FUNCTION_BLOCK "GCS7_E_DCOS"	// FB 43
TITLE = Scale DCOS
//  
//COPYRIGHT:    (C) 2003  BUHLER AG, CH-9240 UZWIL, SWITZERLAND
//
//PRODUCT:      GCS7
//
//TITLE:        Element Control DCOS
//
//-------------------------------------------------------------------------
//
//IDENT:        AUTHOR:             DEPT:                       DATE:
//FB43.2.2      A. Egli             BASE                        09-Apr-2008
//              Disable Alarm 18 Battery Low
//FB43.2.1      A.Egli              CT3                         01-Dec-2005
//              Parameter Upload Change DBD86-->DBD88
//FB43.2.0      A.Egli              CT3                         05-Jan-2005
//              Parameter Upload (uses DB10)
//FB43.1.3      A.Egli              CT3                         13-Apr-2004
//              Copy TotalReady only when Block 1 is read
//FB43.1.2      A.Egli              CT3                         17-Nov-2003
//              - Alarm 90: Fault not DPRemoteControl
//              - Ignor SumFault as long AlarmNr <>0
//FB43.1.1      A. Egli             CT3                         05-Aug-2003
//              Reset Par.HelpFlags.OutIngrActive
//FB43.1.0      A. Egli             CT3                         02-Apr-2003
//              1st Release in S7
//
//-------------------------------------------------------------------------
//
//PURPOSE:      MANUAL : see [DOSxxMAN]
//
//RESTRICTIONS: S7
//
//=======================================================
//Log Message: 
//------------------------------------------------------
//0     = Fault Cannceled
//1..79 = AlarmLC : Alarmnumber see manual of MEAF
//90    = Fault Remote Control
//91    = StPassive
//92    = StDosing
//93    = StEmptied
//94    = Timeout starting
//95    = WrongValue
//96    = Communication fault
//97    = 
//98    = 
//99    = Collected alarm
//
//=======================================================
//StCode:  State               
//------------------------------------------------------
//32   StFault                 
// 1   StPassive               
//41   StPassive.HWStop              StPassive + InHWStop 
//51   StPassive.DPFault             StPassive + DPFault
// 2   StStarting              
// 3   StDosing                
// 9   StEmptying              
//10   StEmptied               
//11   StRefill                
AUTHOR : EA
FAMILY : GCS7LL
NAME : DCOS
VERSION : 2.2
VAR
  StCode : INT ;	//Element state code
  InEnable : BOOL ;	//Enable to run scale
  CmdAbort : BOOL ;	//Abort ingredient
  InLocalControl : BOOL ;	//Local start and abort
  spare23 : BOOL ;
  CmdNewIngr : BOOL ;	//Start new ingredient
  In_Q_ResultIngr : BOOL ;	//Acknowledge resulting
  InEmptying : BOOL ;	//Fully emptying scale hopper
  spare27 : BOOL ;
  CmdOff : BOOL ;	//Pulse to stop scale (manual mode)
  CmdOn : BOOL ;	//Pulse to start scale(manual mode)
  spare33 : BOOL ;	//Ingredient is ready for resulting
  CmdFaultReset : BOOL ;	//Command to reset fault
  InLocal : BOOL ;	//1= Local mode (no fault by start with service switch)
  InManual : BOOL ;	//1= Manual/ 0= Automatic
  InReport : BOOL ;	//Report of all state transitions
  spare37 : BOOL ;
  InHWStop : BOOL ;	//Hardware stop
  OutEnableLocal : BOOL ;
  InSimulation : BOOL ;	//Simulation with DPSim
  Out_F_ResultIngr : BOOL ;	//Announcement resulting ingredient
  OutComFault : BOOL ;	//Communication fault
  OutEmptied : BOOL ;	//Scale hopper is empytied
  OutIngrActive : BOOL ;	//Ingredient is activele
  OutWrongValue : BOOL ;	//Wrong nominal values, rejected by MEAF
  StPassive : BOOL ;	//Element is passive, no ingredient active
  StStarting : BOOL ;	//Scale is starting
  StDosing : BOOL ;	//Scale is dosing
  StEmptying : BOOL ;	//Emptying is active
  StFault : BOOL ;	//Element has a fault
  StEmptied : BOOL ;	//Hopper is emptied
  StWaiting : BOOL ;	//Scale is waiting for next ingredient
  StSuspended : BOOL ;	//Ingredient is suspended
  InRecipeNr : INT ;	//[1..8] Is send to LC
  InWeight : DINT ;	//[DIV] Is send to LC
  OutRecipeNr : INT ;	//Is read from LC
  OutWeight : DINT ;	//[DIV] Ingredient weight, is read from scale
  OutScaleWeight : DINT ;	//[DIV] Scale weight, is read from LC
  spare : DINT ;
  OutDecimalPoint : INT ;	//Is read from LC
  OutLCStep : INT ;	//Is read from LC
  OutAlarmNr : INT ;	//Is read from LC
  OutAlarmNrLog : INT ;	//Last textnumber send to log
  Recipe : STRUCT 	//Recipe Diff Scale (Profibus only)
   InRecipeNr : INT ;	//Recipe to read or write (DIFF only)
   CmdSend : BOOL ;	//1= Send Dataset 136
   CmdRead : BOOL ;	//1= Read Dataset 136
   OutSendDone : BOOL ;	//Send is done
   OutReadDone : BOOL ;	//Read is done
   OutWrongValue : BOOL ;	//MEAF has recipe rejected
   Para : STRUCT 	//DIFF: Pre cutoff weight
    InOutBinNr : INT ;	//Bin number =REC.BIN
    InOutWeightNominal : DINT ;	//[DIV] Target weight  =REC.WTS
    InOutTolPosWeight : INT ;	//[DIV] Tolerance weight positive =REC.TOL+
    InOutTolNegWeight : INT ;	//[DIV] Tolerance weight negative =REC.TOL-
    InOutFineDosingWeight : INT ;	//[DIV] Fine dosing weight =REC.STRT
    InOutCutoffWeight : INT ;	//[DIV] Pre cutoff weight =REC.CUTW
    InOutDosingSpeedFast : INT ;	//[%] Fast dosing speed =REC.FFLO
    InOutDosingSpeedSlow : INT ;	//[%] Slow dosing speed =REC.DFLO
   END_STRUCT ;
  END_STRUCT ;
  Par : STRUCT
   ParObjectNo : INT ;	//Is used for communication with PC, e.g. for message
   ParMsgType : INT ;	//Is used for message (translation of state)
   ParHornCode : INT ;	//Is used by horn module
   ParLogOff : BOOL ;	//Report is off
   ParManual : BOOL ;	//Manual mode without interlocking
   ParPosWeighing : BOOL ;	//1=Positve weighing, 0=Negativ weighing
   ParFilter : STRUCT 	//Filter to alarm 1=Ignore alarm
    SumFault : BOOL ;	//All: de: Sammelalarm
    A05_24VToLow : BOOL ;	//All:
    A07ADRange : BOOL ;
    A08ADCalibration : BOOL ;
    A09ADFunction : BOOL ;
    A10ADSupply : BOOL ;
    A11AnalogInput : BOOL ;
    AxxCommunication : BOOL ;	//A12: Serial Interface ; A14=DPFault
    A13RemoteControl : BOOL ;
    A16Printer : BOOL ;
    A18BatteryLow : BOOL ;
    A20NoStandStill : BOOL ;
    A26Tolerance : BOOL ;
    A30ZeroTara : BOOL ;
    A42Limit : BOOL ;
    A63ProductFlow : BOOL ;
   END_STRUCT ;
   ParIOByteNr : INT ;	//PROFIBUS: Address of first input and output byte Profibus DP
   ParMonTime : INT ;	//After this time the scale must be in the requested state (New)
   Spare90 : DINT ;
   Spare94 : DINT ;
   OutMonTime : INT ;
   HelpFlags : STRUCT 	//Aux. signal to retry fault message
    OutFaultResetDone : BOOL ;
    OutTestNewAlarm : BOOL ;
    OutFlagFaultResetDone : BOOL ;
    OutAlarmTimeOut : BOOL ;
    spare : BOOL ;	//Help flag for immediate stop
    OutRelevantFault : BOOL ;
    OutNoAlarm : BOOL ;	//Alarmnumber 0 is read form LC
    OutComFaultRead : BOOL ;
    OutComFaultSend : BOOL ;
    OutIngrActive : BOOL ;
   END_STRUCT ;
   Command : STRUCT 	//Command for LC, is send to LC
    Start : BOOL ;	//de: Start
    Abort : BOOL ;	//de: Abbruch
    ControlByDP : BOOL ;	//de: Bedienung über Profibus DP
    spare03 : BOOL ;
    spare04 : BOOL ;
    spare05 : BOOL ;
    Emptying : BOOL ;	//de: Entleeren / Charge beenden
    AcceptTotalReady : BOOL ;	//de: Quittierung neue Werte Bereit
    AcceptStart : BOOL ;	//de: Quittierung 24V Start/Stop Signal
    AcceptAbort : BOOL ;	//de: Quittierung 24V Abbruch Signal
    spare20 : BYTE ;
    CommandReady : BOOL ;	//de: Steuersignale gültig
    spare41 : BOOL ;
    spare42 : BOOL ;
    spare43 : BOOL ;
    spare44 : BOOL ;
    ResetAlarm : BOOL ;	//de: Alarm löschen
    NewSendData : BOOL ;	//de: Aenderung Sendedaten
    AcceptNewRcvData : BOOL ;	//de: Quittierung Aenderung Empfangsdatensatz
   END_STRUCT ;
   Status : STRUCT 	//MEAF DIFF
    Operation : BOOL ;	//de: Betrieb
    spare01 : BOOL ;
    ReadyDosing : BOOL ;	//de: Dosierbereit
    FastDosing : BOOL ;	//de: Grobdosieren
    SlowDosing : BOOL ;	//de: Feindosieren
    Emptying : BOOL ;	//de: Entleerung aktiv
    EmptyingDone : BOOL ;	//de: Entleeren ausgefüht
    TotalReady : BOOL ;	//de: Total erreicht
    Start : BOOL ;	//de: Start/Stop 24V
    Abort : BOOL ;	//de: Abbruch 24V
    spare20 : BYTE ;
    spare30 : BOOL ;
    spare31 : BOOL ;
    spare32 : BOOL ;	//de: Stuerung Remote
    RemoteControlDP : BOOL ;	//de: Sollwertvorgabe Remote
    WrongValue : BOOL ;	//de: Falscher Sollwert
    SumFault : BOOL ;	//de: Sammelalarm
    AcceptNewSendData : BOOL ;	//de: Quittierung Aenderung Sendedaten
    NewRcvData : BOOL ;	//de: Aenderung Empfangsdaten
   END_STRUCT ;
  END_STRUCT ;
END_VAR
VAR_TEMP
  tmpLOGvalue : WORD ;	//LOG value
  tmpCommand : INT ;
  tmpReport : BOOL ;	//Global LOG all
  tmpFault : BOOL ;
  tmpLocal : BOOL ;
  tmpOn : BOOL ;
  tmpOff : BOOL ;
  tmpSeqStopDUMP : BOOL ;
  tmpWeight : DINT ;
  tmpLenDyn : DINT ;
  tmpImmediateStop : BOOL ;
  tmpFilter : ARRAY  [0 .. 100 ] OF BOOL ;
  tmpAlarmDIFF : STRUCT 	//Is read from DIFF with command d
   DepotEmpty : BOOL ;	//Surge hopper empty (not on collect alarm) --> alarm 34
   ScaleEmpty : BOOL ;	//de: Leerstand Waage (no product)
   Discharger : BOOL ;	//DIFF a2 Frequency converter or feeding drive -->alarm 25
   Tolerance : BOOL ;	//DIFF a2 Tolerance --> alarm 26
   SumFault : BOOL ;	//de: Sammelalarm ab V26A
   TaraPos : BOOL ;	//DIFF a1 n.w.  -->alarm 30
   ADConverter : BOOL ;	//DIFF a1 AD converter--> alarm 9
   Reading : BOOL ;	//DIFF a1 Measuring fault --> alarm 27
  END_STRUCT ;
  tmpAddr : WORD ;
  tmpReturn : INT ;
  DPData : STRUCT
   StatusCommand : DWORD ;
   NrSndDataSet : BYTE ;	//de: Nummer Sendedatensatz
   IdxSndDataSet : BYTE ;	//de: Index Sendedatensatz
   NrRcvDataSet : BYTE ;	//de: Nummer Empfangsdatensatz
   IdxRcvDataSet : BYTE ;	//de: Index Empfangsdatensatz
   Data : STRUCT
    Value8 : DINT ;
    Value12 : DINT ;
    Value16 : DINT ;
    Value20 : BYTE ;
    Value21 : BYTE ;
    Value22 : BYTE ;
    Value23 : BYTE ;
   END_STRUCT ;
  END_STRUCT ;
  tmpTotalReady : BOOL ;
END_VAR
BEGIN
NETWORK
TITLE =  Start Global
      L     90;
      T     #tmpLenDyn;	//--> Len dynamic data in byte
NETWORK
TITLE = Filter
      LAR1  P##tmpFilter;
      L     0;
      T     D [AR1,P#0.0];	//tmpFilter[00..31]
      T     D [AR1,P#0.0];	//tmpFilter[32..63]
      T     D [AR1,P#0.0];	//tmpFilter[64..95]
      SET;	//[1.2]
      =     #tmpFilter[0];
      A     #Par.ParFilter.A05_24VToLow;
      =     #tmpFilter[5];
      A     #Par.ParFilter.A07ADRange;
      =     #tmpFilter[7];
      A     #Par.ParFilter.A08ADCalibration;
      =     #tmpFilter[8];
      A     #Par.ParFilter.A09ADFunction;
      =     #tmpFilter[9];
      A     #Par.ParFilter.A10ADSupply;
      =     #tmpFilter[10];
      A     #Par.ParFilter.A11AnalogInput;
      =     #tmpFilter[11];
      A     #Par.ParFilter.AxxCommunication;
      =     #tmpFilter[12];
      =     #tmpFilter[14];
      A     #Par.ParFilter.A13RemoteControl;
      =     #tmpFilter[13];
      A     #Par.ParFilter.A16Printer;
      =     #tmpFilter[16];
      SET;
      =     #tmpFilter[18];	//[2.2] Battery Low
      A     #Par.ParFilter.A20NoStandStill;
      =     #tmpFilter[20];
      A     #Par.ParFilter.A26Tolerance;
      =     #tmpFilter[26];
      A     #Par.ParFilter.A30ZeroTara;
      =     #tmpFilter[30];
      A     #Par.ParFilter.A42Limit;
      =     #tmpFilter[42];
      A     #Par.ParFilter.A63ProductFlow;
      =     #tmpFilter[63];
NETWORK
TITLE = PC Control
//=== Test Object number =====================
      L     "SYS_DirectCtrlDB".PC.ObjectNo;	//PCControl.ObjectNo
      L     #Par.ParObjectNo;	//Input ObjectNo
      <>I;
      JC    Ctrl;
//=== Test OType      ========================
      L     1043;	//Input object type
      L     "SYS_DirectCtrlDB".PC.ObjectType;	//PCControl.ObjectType
      <>I;
      JC    Ctrl;
//=== Test Handshake =========================
      A     "SYS_DirectCtrlDB".PC.Hsk.FExamine;	//Handshake.FExamine
      JC    pExa;
      A     "SYS_DirectCtrlDB".PC.Hsk.FDefineCmd;	//Handshake.FDefineCmd
      JC    pCmd;
      A     "SYS_DirectCtrlDB".PC.Hsk.FDefinePara;	//Handshake.FDefinePara
      JC    pPar;
pIni: L     2;	//FcInit
      UC    "SYS_DirectCtrl";
      JU    Ctrl;
// Write parameter 
pPar: LAR1  P#DBX 58.0;
      L     P##Par;
      L     DW#16#FFFFF;
      AD;
      +AR1;
      L     DBD [AR1,P#12.0];
      T     #Par.ParMonTime;
//Write new commands from PC to Interface of group 
pCmd: A     "SYS_DirectCtrlDB".PC.Cmd1[1];	//Cmd1[1]  =CmdAbort
      S     #CmdAbort;
      A     "SYS_DirectCtrlDB".PC.Cmd1[6];	//Cmd1[2]  =CmdEmptyingOn
      S     #InEmptying;
      A     "SYS_DirectCtrlDB".PC.Cmd2[6];	//Cmd1[2]  =CmdEmptyingOff
      R     #InEmptying;
      A     "SYS_DirectCtrlDB".PC.Cmd1[4];	//Cmd1[4]  =CmdNewIngr
      S     #CmdNewIngr;
      R     #InEmptying;
      A     "SYS_DirectCtrlDB".PC.Cmd1[5];	//Cmd1[5]  =Cmd_Q_ResultIngr
      S     #In_Q_ResultIngr;
      A     "SYS_DirectCtrlDB".PC.Cmd1[8];	//Cmd1[8]  =CmdOff
      S     #CmdOff;
      A     "SYS_DirectCtrlDB".PC.Cmd1[9];	//Cmd1[9]  =CmdOn
      S     #CmdOn;
      A     "SYS_DirectCtrlDB".PC.Cmd1[11];	//Cmd1[11]=CmdFaultReset
      S     #CmdFaultReset;
      A     "SYS_DirectCtrlDB".PC.Cmd1[13];	//Cmd1[13]=CmdManualOn
      S     #InManual;
      A     "SYS_DirectCtrlDB".PC.Cmd2[13];	//Cmd2[13]=CmdManualOff
      R     #InManual;
      A     "SYS_DirectCtrlDB".PC.Cmd1[14];	//Cmd1[14]=CmdReportOn
      S     #InReport;
      A     "SYS_DirectCtrlDB".PC.Cmd2[14];	//Cmd2[14]=CmdReportOff
      R     #InReport;
//Define Value
      AN    "SYS_DirectCtrlDB".PC.Hsk.FDefineValue;	// PC.Hsk.FDefineValue
      ON    #InManual;
      JC    pIni;
      LAR1  P#DBX 58.0;
      L     DBW [AR1,P#6.0];
      T     #InRecipeNr;
      L     DBD [AR1,P#8.0];
      T     #InWeight;
      JU    pIni;
pExa: TAR2;	//Address Dynamic datas
      T     "SYS_DirectCtrlDB".GC.InDynAddr;	//-->PCControl.GC.InDynAddr
      L     #tmpLenDyn;	//Length Dynamic datas
      T     "SYS_DirectCtrlDB".GC.InDynLen;	//-->PCControl.GC.InDynLen
      L     0;
      T     "SYS_DirectCtrlDB".GC.InParaAddr;	//-->PCControl.GC.InParaAddr
      T     "SYS_DirectCtrlDB".GC.InParaLen;	//-->PCControl.GC.InParaLen
      L     1;	//Code FcExamine
      UC    "SYS_DirectCtrl";
      L     10;	//Revision
      T     "SYS_DirectCtrlDB".GC.Revision;
Ctrl: NOP   0;
NETWORK
TITLE = (Profibus) Read data
//**********************************
//(Profibus)
//**********************************
      L     #Par.ParIOByteNr;
      T     #tmpAddr;
      A     #InSimulation;
      JC    rSim;
      CALL  "SIEMENS_DPRD_DAT" (
           LADDR                    := #tmpAddr,
           RET_VAL                  := #tmpReturn,
           RECORD                   := #DPData);
      L     #tmpReturn;
      L     0;
      <>I;
      =     #Par.HelpFlags.OutComFaultRead;
      JC    rcv0;
      JU    rDP;
//read from Simulation
rSim: R     #Par.HelpFlags.OutComFaultRead;
      A     "GCS7_Gr_SimDPtoImage";
      L     P#I 0.0;
      JC    rDB1;
      OPN   "TEST_IOSimuliInput";
      L     P#DBX 0.0;
rDB1: L     #Par.ParIOByteNr;
      SLD   3;
      +D;
      LAR1;
      L     D [AR1,P#0.0];
      T     #DPData.StatusCommand;
      L     B [AR1,P#4.0];
      T     #DPData.NrSndDataSet;
      L     B [AR1,P#5.0];
      T     #DPData.IdxSndDataSet;
      L     B [AR1,P#6.0];
      T     #DPData.NrRcvDataSet;
      L     B [AR1,P#7.0];
      T     #DPData.IdxRcvDataSet;
      L     D [AR1,P#8.0];
      T     #DPData.Data.Value8;
      L     D [AR1,P#12.0];
      T     #DPData.Data.Value12;
      L     D [AR1,P#16.0];
      T     #DPData.Data.Value16;
      L     B [AR1,P#20.0];
      T     #DPData.Data.Value20;
      L     B [AR1,P#21.0];
      T     #DPData.Data.Value21;
      L     B [AR1,P#22.0];
      T     #DPData.Data.Value22;
      L     B [AR1,P#23.0];
      T     #DPData.Data.Value23;
//==Copy Status===============
rDP:  L     #DPData.NrRcvDataSet;
      L     0;
      ==I;
      JC    R001;
      A     #Par.Status.TotalReady;	//[1.3]
      =     #tmpTotalReady;	//[1.3]
      CALL  "SIEMENS_BLKMOV" (
           SRCBLK                   := #DPData.StatusCommand,
           RET_VAL                  := #tmpReturn,
           DSTBLK                   := #Par.Status);
      A     #tmpTotalReady;	//[1.3]
      =     #Par.Status.TotalReady;	//[1.3]
      AN    #Par.Status.NewRcvData;
      A     #InSimulation;
      JC    rcv0;
//===============================
//Answer Dataset 001
      L     #DPData.NrRcvDataSet;
      L     1;
      <>I;
      JC    r11;	//[2.0]
      CALL  "SIEMENS_BLKMOV" (
           SRCBLK                   := #DPData.StatusCommand,
           RET_VAL                  := #tmpReturn,
           DSTBLK                   := #Par.Status);	//[1.3]
      AN    #Par.HelpFlags.OutIngrActive;
      JC    rJ4;
      L     #DPData.Data.Value8;
      T     #OutWeight;
rJ4:  L     #DPData.Data.Value12;
      T     #OutScaleWeight;
      L     #DPData.Data.Value20;
      T     #OutDecimalPoint;
      L     #DPData.Data.Value21;
      T     #OutRecipeNr;
      L     #DPData.Data.Value22;
      T     #OutLCStep;
//Reset old alarm flags with CmdFaultReset
      A     #Par.HelpFlags.OutFlagFaultResetDone;
      A     "SYS_Pulse1000ms";
      R     #Par.HelpFlags.OutFlagFaultResetDone;
      R     #Par.HelpFlags.OutFaultResetDone;
      S     #Par.HelpFlags.OutTestNewAlarm;
      L     #DPData.Data.Value23;	//[1.2]
      L     0;	//[1.2]
      <>I;	//[1.2]
      O     #Par.ParFilter.SumFault;	//[1.2]
      =     #tmpFilter[0];	//[1.2]
      L     0;
      L     #DPData.Data.Value23;
      ==I;
      =     #Par.HelpFlags.OutNoAlarm;
//  keep old alalrm number
      A     #Par.HelpFlags.OutNoAlarm;
      A     #Par.HelpFlags.OutRelevantFault;
      AN    #Par.HelpFlags.OutTestNewAlarm;
      AN    #InLocal;
      AN    #InManual;
      JC    rA1;
      T     #OutAlarmNr;
rA1:  NOP   0;
      JU    R11;	//[2.0]   
//===============================
//[7.0]--> LC Parameter 
//Reading dataset 11
R11:  L     "SYS_DirectCtrlLCDB".PC.ObjectNo;
      L     #Par.ParObjectNo;
      <>I;
      JC    R127;
      AN    "SYS_DirectCtrlLCDB".PC.Hsk.FExamineFirst;
      AN    "SYS_DirectCtrlLCDB".PC.Hsk.FExamineNext;
      JC    R127;
// -- Start Reading with Dataset 11
      L     11;
      T     #DPData.NrRcvDataSet;
      L     253;	//First
      A     "SYS_DirectCtrlLCDB".PC.Hsk.FExamineFirst;
      JC    rLC9;
      L     254;	//Next
rLC9: T     #DPData.IdxRcvDataSet;
      JU    rcv0;
//---Answer  dataset 11 ---
//---Answer  dataset 12 ---
r11:  L     #DPData.NrRcvDataSet;
      L     11;
      <>I;
      JC    rLCB;
// Answer Dataset 11
      L     '  ';
      T     "SYS_DirectCtrlLCDB".PC.Value[1];
      L     #DPData.Data.Value8;
      T     DB10.DBD 60;
      L     #DPData.Data.Value12;
      T     DB10.DBD 64;
      L     #DPData.Data.Value16;
      T     DB10.DBD 68;
      L     #DPData.Data.Value20;
      SLD   24;
      L     #DPData.Data.Value21;
      SLD   16;
      OD;
      L     #DPData.Data.Value22;
      SLD   8;
      OD;
      L     #DPData.Data.Value23;
      OD;
      T     DB10.DBD 72;
      L     #DPData.IdxRcvDataSet;
      L     255;
      ==I;
      JC    rLCE;
      S     "SYS_DirectCtrlLCDB".GC.Set11Done;
      L     12;
      T     #DPData.NrRcvDataSet;
      L     0;
      T     #DPData.IdxRcvDataSet;
      JU    rcv0;	//--> Read dataset 12
// Answer Dataset 12
rLCB: L     #DPData.NrRcvDataSet;
      L     12;
      <>I;
      JC    r127;
      L     #DPData.Data.Value8;
      T     DB10.DBD 76;
      L     #DPData.Data.Value12;
      T     DB10.DBD 80;
      L     #DPData.Data.Value16;
      T     DB10.DBD 84;
      L     #DPData.Data.Value20;
      SLD   24;
      L     #DPData.Data.Value21;
      SLD   16;
      OD;
      L     #DPData.Data.Value22;
      SLD   8;
      OD;
      L     #DPData.Data.Value23;
      OD;
      T     DB10.DBD 88;
      AN    "SYS_DirectCtrlLCDB".GC.Set11Done;
      JC    R127;
rLCE: L     12;
      CALL  "SYS_DirectCtrl";
      JU    R127;
//<--[2.0]
//===============================
//Answer  dataset 127
r127: L     #DPData.NrRcvDataSet;
      L     127;
      <>I;
      JC    r128;
      JU    R128;
//===============================
//Answer  dataset 128
r128: L     #DPData.NrRcvDataSet;
      L     128;
      <>I;
      JC    r136;
      JU    R001;
//===============================
//Answer  dataset 136
r136: L     #DPData.NrRcvDataSet;
      L     136;
      <>I;
      JC    R001;	// =no valide answer read dataset 001
      L     #Recipe.InRecipeNr;
      L     #DPData.IdxRcvDataSet;
      ==I;
      JCN   R001;
      S     #Recipe.OutReadDone;
      R     #Recipe.CmdRead;
      CALL  "SIEMENS_BLKMOV" (
           SRCBLK                   := #DPData.Data,
           RET_VAL                  := #tmpReturn,
           DSTBLK                   := #Recipe.Para);
      L     #DPData.Data.Value22;
      T     #Recipe.Para.InOutDosingSpeedFast;
      L     #DPData.Data.Value23;
      T     #Recipe.Para.InOutDosingSpeedSlow;
      JU    R001;
//===============================
//Read Dataset 001
R001: L     1;
      T     #DPData.NrRcvDataSet;
      L     0;
      T     #DPData.IdxRcvDataSet;
      A     #Par.HelpFlags.OutFaultResetDone;
      AN    "SYS_Pulse1000ms";
      S     #Par.HelpFlags.OutFlagFaultResetDone;
      JU    rcv0;
//===============================
//Read Dataset 127
R127: L     127;
      T     #DPData.NrRcvDataSet;
      L     0;
      T     #DPData.IdxRcvDataSet;
      JU    rcv0;
//===============================
//Read Dataset 128
R128: JU    R136;
      JU    rcv0;
//===============================
//Read Dataset 136
R136: AN    #Recipe.CmdRead;
      JC    R001;
      L     136;
      T     #DPData.NrRcvDataSet;
      L     #Recipe.InRecipeNr;
      T     #DPData.IdxRcvDataSet;
rcv0: NOP   0;
      A     #Par.HelpFlags.OutComFaultRead;
      O     #Par.HelpFlags.OutComFaultSend;
      =     #OutComFault;
      NOP   0;
NETWORK
TITLE = Local Control
// ---Abort
      A     #Par.Status.Abort;
      A     #InLocalControl;
      S     #CmdAbort;
// -- Start Ingredient
      A     #Par.Status.Start;
      AN    #Par.Command.AcceptStart;
      A     #Par.Status.ReadyDosing;
      A     #InLocalControl;
      AN    #OutIngrActive;
      S     #CmdNewIngr;
      S     #OutEnableLocal;
// -- Start Local
      A     #Par.Status.Start;
      AN    #Par.Command.AcceptStart;
      AN    #OutEnableLocal;
      S     #OutEnableLocal;
      JC    aiL1;
// -- Stop Local
      A     #Par.Status.Start;
      AN    #Par.Command.AcceptStart;
      A     #OutEnableLocal;
      AN    #CmdNewIngr;
      O     #Par.Status.Abort;
      ON    #InLocalControl;
      O;
      AN    #OutIngrActive;
      AN    #CmdNewIngr;
      R     #OutEnableLocal;
aiL1: NOP   0;
NETWORK
TITLE =  All State Init
      NOP   0;
//===Global Group Orders===
      A     "GCS7_Gr_OutManualOn";	//Gr.OutManualOn
      S     #InManual;
      A     "GCS7_Gr_OutManualOff";	//Gr.OutManualOff
      R     #InManual;
      A     #InManual;
      S     "GCS7_Gr_InManual";	//Gr.InManualMode
      A     "GCS7_Gr_OutFaultReset";	//Gr.OutOutFaultReset
      O     #CmdAbort;
      S     #CmdFaultReset;
//---Report is on---
      A     "GCS7_Gr_OutReportAll";	//Gr.OutReportAll
      O     #InReport;
      =     #tmpReport;
//---Local---
      A     #InLocal;
      AN    #InManual;
      =     #tmpLocal;
//---Enable---
// tmpOff
      AN    #InEnable;
      AN    #Par.ParManual;	// 2C: U -> UN
      A     #InManual;
      O;
      AN    #InEnable;
      AN    #InManual;
      O     #CmdOff;
      O     #tmpLocal;
      O(;
      A     #InLocalControl;
      AN    #OutEnableLocal;
      );
      O     #InHWStop;
      =     #tmpOff;
      R     #OutEnableLocal;
//---On---
      AN    #InManual;
      O     #CmdOn;
      AN    #tmpOff;
      =     #tmpOn;
//--- Init in local mode  
      AN    #tmpLocal;
      JC    alJL;
      R     #OutComFault;
alJL: NOP   0;
//--- Fault   
      LAR1  P##tmpFilter;
      L     #OutAlarmNr;
      +AR1;	//Pointer to #tmpFilter[OutAlarmNumber]
      L     #OutAlarmNr;
      L     0;
      <>I;
      AN    L [AR1,P#0.0];	//#tmpFilter[OutAlarmNumber]
      O;
      A     #Par.Status.SumFault;
      AN    #tmpFilter[0];
      =     #Par.HelpFlags.OutRelevantFault;
      A     #Par.HelpFlags.OutRelevantFault;
      O     #OutComFault;
      O     #OutWrongValue;
      ON    #Par.Status.RemoteControlDP;	//[1.2]
      AN    #tmpLocal;
      =     #tmpFault;
//-- Ingredient done
      A     #Out_F_ResultIngr;
      A     #In_Q_ResultIngr;
      R     #OutIngrActive;
      A     #CmdAbort;
      O     #Par.Status.TotalReady;
      A     #OutIngrActive;
      AN    #In_Q_ResultIngr;
      =     #Out_F_ResultIngr;
//-----------------------
      A     #CmdNewIngr;
      R     #Out_F_ResultIngr;
      R     #In_Q_ResultIngr;
      R     #OutIngrActive;
      R     #Par.HelpFlags.OutIngrActive;	//[1.1]
//--Reset Actual weight during start
      A     #Par.Status.FastDosing;
      O     #Par.Status.SlowDosing;
      O     #Out_F_ResultIngr;
      S     #Par.HelpFlags.OutIngrActive;
      AN    #CmdNewIngr;
      JC    alJ2;
      L     0;
      T     #OutWeight;
//--- Recipe
alJ2: A     #Recipe.CmdRead;
      R     #Recipe.OutReadDone;
      A     #Recipe.CmdSend;
      R     #Recipe.OutSendDone;
//---Abort if Local
      A     #tmpLocal;
      A     #OutIngrActive;
      S     #CmdAbort;
      R     #CmdNewIngr;
      A     #Par.Status.ReadyDosing;
      A     #tmpLocal;
      R     #OutIngrActive;
NETWORK
TITLE = Monitoring [6.0]
//Monitoring Time [6.0]
      A     #StPassive;
      O     #CmdFaultReset;
      R     #Par.HelpFlags.OutAlarmTimeOut;	//[6.0]
      AN    #StStarting;	//[6.0]
      JC    mtJ0;	//[6.0]
      ON    "GCS7_Gr_OutTick200ms";	//[6.0]
      JC    mtJ1;	//[6.0]
      L     #Par.OutMonTime;	//[6.0]
      +     -2;	//[6.0]
      T     #Par.OutMonTime;	//[6.0]
      L     0;	//[6.0]
      >=I;	//[6.0]
      JC    mtJ1;	//[6.0]
      S     #Par.HelpFlags.OutAlarmTimeOut;	//[6.0]
      JU    mtJ1;	//[6.0]
mtJ0: L     #Par.ParMonTime;	//[6.0]
      T     #Par.OutMonTime;	//[6.0]
mtJ1: NOP   0;
NETWORK
TITLE = States
//===State machine===
      A     #StPassive;
      JC    S0;
      A     #StStarting;
      JC    S1;
      A     #StDosing;
      JC    S2;
      A     #StEmptying;
      JC    S3;
      A     #StFault;
      JC    S4;
      A     #StEmptied;
      JC    S5;
      A     #StWaiting;
      JC    S6;
      A     #StSuspended;
      JC    S7;
      S     #StPassive;	//Init
NETWORK
TITLE = StPassive
//Transition to StPassive
//Transition
xxS0: S     #StPassive;
      JU    LOGX;
//----------------------------------------------
//Logic
//Condition for StFault
S0:   A     #tmpFault;
      R     #StPassive;
      JC    xxS4;
//StEmptying
      AN    #tmpOff;
      A     #InEmptying;
      R     #StPassive;
      JC    xxS3;
//Condition for StStarting
      AN    #Par.Command.Abort;
      A     #CmdNewIngr;
      AN    #tmpOff;
      A     #Par.Status.ReadyDosing;
      AN    #Par.Status.TotalReady;
      AN    #Par.Command.AcceptTotalReady;
      R     #StPassive;
      JC    xxS1;
      JU    OUT;
NETWORK
TITLE =  STARTING
// Any Transition
//Transition
xxS1: S     #StStarting;
      S     #OutIngrActive;
      R     #CmdNewIngr;
      R     #OutEmptied;
      JU    OUT;
//----------------------------------------------
//Logic
S1:   NOP   0;
//Condition for StFault
      A     #tmpFault;
      O     #Par.HelpFlags.OutAlarmTimeOut;	//Monitoring Time [6.0]
      R     #StStarting;
      JC    xxS4;
//-- Transition to StDosing --         
      A     #Par.Status.Operation;
      AN    #OutComFault;	//[1.2]
      R     #StStarting;
      JC    xxS2;
//Condition for StSuspended
      A     #tmpOff;
      R     #StStarting;
      JC    xxS7;
//Condition for StWaiting
      AN    #OutIngrActive;
      R     #StStarting;
      JC    xxS6;
      JU    OUT;
NETWORK
TITLE =  DOSING
//Transition
//----------------------------------------------
xxS2: SET;
      S     #StDosing;
      JU    LOGX;
//----------------------------------------------
//Condition for StWaiting
S2:   AN    #OutIngrActive;
      R     #StDosing;
      JC    xxS6;
//Condition for StSuspended
      AN    #Par.Command.Start;
      O     #OutComFault;	//[1.2]
      R     #StDosing;
      JC    xxS7;
//Monitoring Time [6.0]
      A     #Par.HelpFlags.OutAlarmTimeOut;	//[6.0]
      R     #StDosing;	//[6.0]
      JC    xxS4;	//[6.0]
//Condition for Fault
      A     #tmpFault;
      R     #StDosing;
      JC    xxS4;
      JU    OUT;
NETWORK
TITLE =  FAULT
      NOP   0;
//Fault cancelled
S4:   A     #Par.HelpFlags.OutTestNewAlarm;
      AN    #tmpFault;
      O     #tmpLocal;
      JC    S4xx;
      A     #Par.HelpFlags.OutTestNewAlarm;	//[2.3] Relog fault
      A     #tmpFault;	//[2.3]
      JC    xxS4;	//[2.3]
      JU    OUT;
//Transition to StSuspended
S4xx: A     #OutIngrActive;
      R     #StFault;
      S     #StSuspended;
      JC    LOG2;	//-->//Message ('fault cancelled')
//Transition to StWaiting 
      R     #StFault;
      S     #StWaiting;
      JU    LOG2;	//-->//Message ('fault cancelled')
NETWORK
TITLE =  StEmptying
//Transition
//----------------------------------------------
xxS3: S     #StEmptying;
      JU    OUT;
//----------------------------------------------
// Condition for fault
S3:   A     #tmpFault;
      R     #StEmptying;
      JC    xxS4;
//Condition for emptied
      L     #OutScaleWeight;
      L     0;
      ==I;
      O     #Par.Status.EmptyingDone;
//     O     #Par.Status.TotalReady
      ON    #Par.ParPosWeighing;
      R     #StEmptying;
      JC    xxS5;	//-->StEmptied
//[4.0->] Back to Stopped if not emptying
      AN    #InEmptying;
      R     #StEmptying;	//avoid setting of OutEmptied
      R     #InEmptying;
      JC    xxS0;	//[<-4.0]
      JU    OUT;
NETWORK
TITLE =  StEmptied
//Condition for fault
//Transition
//----------------------------------------------
xxS5: S     #StEmptied;
      S     #OutEmptied;
      JU    LOGX;
//----------------------------------------------
S5:   A     #tmpFault;
      R     #StEmptied;
      JC    xxS4;
//Condition for Starting/Waiting
      A     #CmdNewIngr;
      R     #StEmptied;
      JC    xxS6;
//Condition for Stopped
      AN    #InEmptying;
      O     #tmpOff;
      R     #StEmptied;
      JC    xxS0;
      JU    OUT;
NETWORK
TITLE = StWaiting
//Transition
xxS6: S     #StWaiting;
      JU    OUT;
//----------------------------------------------
//Condition for fault
S6:   A     #tmpFault;
      R     #StWaiting;
      JC    xxS4;
//Condidition for StPassive
      A     #tmpLocal;
      ON    #Par.ParPosWeighing;
      R     #StWaiting;
      JC    xxS0;
//Condition for Starting
      A     #CmdNewIngr;
      AN    #Par.Command.Abort;
      AN    #Par.Status.TotalReady;
      AN    #Par.Command.AcceptTotalReady;
      R     #StWaiting;
      JC    xxS1;
//Condition for StEmptying
      A     #InEmptying;
      R     #StWaiting;
      JC    xxS3;
      JU    OUT;
NETWORK
TITLE = StSuspended
//Transition
xxS7: S     #StSuspended;
      JU    OUT;
//----------------------------------------------
//Condition for fault
S7:   A     #tmpFault;
      R     #StSuspended;
      JC    xxS4;
//Condition for Starting
      A     #Par.Command.Start;
      AN    #OutComFault;	//[1.2]
      A     #OutIngrActive;
      AN    #CmdAbort;
      R     #StSuspended;
      JC    xxS1;
//Condition for StWaiting
      AN    #OutIngrActive;
      R     #StSuspended;
      JC    xxS6;
      JU    OUT;
NETWORK
TITLE = LOG
////[5.0] Alarmnummer
xxS4: S     "GCS7_Gr_InFaultFlag";	//Gr.InFaultFlag
      S     #StFault;
//Horn On
      CALL  "SYS_Horn_Code" (
           FcCode                   := 1,
           ParObjectType            := 1040,
           ParObjectNo              := #Par.ParObjectNo,
           ParHornCode              := #Par.ParHornCode);
//Alarm Communication
      L     B#(1, 96);
      A     #OutComFault;
      JC    LOG;
//Tiemout
      A     #Par.HelpFlags.OutAlarmTimeOut;
      L     B#(1, 97);	// Message ('fault timeout')
      JC    LOG;
//Alarm-Nr 1..80
      L     0;
      L     #OutAlarmNr;
      ==I;
      JC    LOG1;
      L     B#(1, 0);
      OW;
      JU    LOG;	//Alarms 1..80
//Fault Remote Control
LOG1: L     B#(1, 90);	// Message ('fault DP Mode')   //[1.2]
      AN    #Par.Status.RemoteControlDP;	//[1.2]
      JC    LOG;	//[1.2]
//Wrong Value
      A     #OutWrongValue;
      L     B#(1, 95);	// Message ('fault wrong value')
      JC    LOG;
//Collected Alarm
      L     B#(1, 99);	// Message ('fault collected alarm')
      JU    LOG;
//Fault Cancelled
LOG2: L     B#(4, 0);	// Message ('fault collected alarm')
      JU    LOG;
//===============================================
//State Transition
LOGX: AN    #tmpReport;
      JC    OUT;
      A     #StPassive;
      L     B#(4, 91);	//Message ('Passive')
      JC    LOG;
      A     #StDosing;
      L     B#(4, 92);	//Message ('Dosing')
      JC    LOG;
      A     #StEmptied;
      L     B#(4, 93);	//Message ('Waiting')
      JC    LOG;
      A     #StEmptied;
      L     B#(4, 94);	//Message ('Emptied')
      JC    LOG;
      JU    OUT;
LOG:  A     #Par.ParLogOff;	//---Set LOG Message
      JC    OUT;
      T     #tmpLOGvalue;
      L     W#16#FF;
      AW;
      T     #OutAlarmNrLog;
      CALL  "GCS7_LogConvert" (
           ObjectNo                 := #Par.ParObjectNo,
           MsgType                  := #Par.ParMsgType,
           ClassMsgTxt              := #tmpLOGvalue,
           OType                    := 1043);	//LOG Message Converter / Entry / Contains Class and TextNo
OUT:  NOP   0;
NETWORK
TITLE = Prepare Command for MEAF
      NOP   0;
//==============================
//Abort
      A     #CmdNewIngr;
      O     #CmdAbort;
      O     #tmpLocal;
      AN    #Par.Status.TotalReady;
      A     #Par.Status.Operation;
      AN    #Par.Status.ReadyDosing;
      =     #Par.Command.Abort;
      AN    #Par.Status.Operation;
      O     #Par.Status.ReadyDosing;
      AN    #OutIngrActive;
      R     #CmdAbort;
//==============================
//  Start/Stop
      A     #StSuspended;
      A     #tmpOn;
      O     #StStarting;
      O     #StDosing;
      AN    #tmpOff;
      AN    #Par.Status.TotalReady;
      AN    #Par.Command.Abort;
      =     #Par.Command.Start;
//==============================
      SET;
      =     #Par.Command.ControlByDP;
//==============================
      L     #OutLCStep;
      L     1;
      >I;
      O     #StEmptying;
      A     #InEmptying;
      =     #Par.Command.Emptying;
//==============================
      A     #CmdAbort;
      O     #CmdFaultReset;
      AN    #Par.Status.AcceptNewSendData;
      S     #Par.Command.ResetAlarm;
      R     #CmdFaultReset;
      A     #Par.Status.AcceptNewSendData;
      A     #Par.Command.ResetAlarm;
      R     #Par.Command.ResetAlarm;
      S     #Par.HelpFlags.OutFaultResetDone;
//==============================
      A     #In_Q_ResultIngr;
      ON    #OutIngrActive;
      A     #Par.Status.TotalReady;
      =     #Par.Command.AcceptTotalReady;
//==============================
      A     #Par.Status.Start;
      =     #Par.Command.AcceptStart;
//==============================
      A     #Par.Status.Abort;
      =     #Par.Command.AcceptAbort;
//==============================
      L     #OutLCStep;
      L     8;
      <>I;
      O     "SYS_Pulse1000ms";
      ON    #Par.Status.EmptyingDone;
      =     #Par.Command.CommandReady;
//==============================
      A     #Par.Status.NewRcvData;
      =     #Par.Command.AcceptNewRcvData;
//==============================
      AN    #Par.Status.AcceptNewSendData;
      =     #Par.Command.NewSendData;
NETWORK
TITLE = Global End
      SET;	//---Clear commands
      R     #CmdOn;
      R     #Par.HelpFlags.OutTestNewAlarm;
      R     #CmdOff;
      NOP   0;
//--Output for group 
      A     #StFault;
      S     "GCS7_Gr_InFault";	// Gr.InFault
NETWORK
TITLE = (Profibus) Send Data
//Test Send Dataset 000 done
      L     #DPData.NrSndDataSet;
      L     0;
      <>I;
      JC    s128;
      JU    S128;	//-->send 128
//------------------------------------------------
//Test Send Dataset 128 done
s128: L     #DPData.NrSndDataSet;
      L     128;
      <>I;
      JC    s136;
      A     #Par.Status.WrongValue;
      =     #OutWrongValue;
      JU    S136;	//-->Send 136
//------------------------------------------------
//Test Send Dataset 129,136 done
s136: L     #DPData.NrSndDataSet;
      L     136;
      <>I;
      JC    S000;
      L     #DPData.IdxSndDataSet;
      L     #Recipe.InRecipeNr;
      ==I;
      JCN   S128;	//-->Send 128
      AN    #Par.Status.WrongValue;
      R     #Recipe.CmdSend;
      =     #Recipe.OutSendDone;
      A     #Par.Status.WrongValue;
      =     #Recipe.OutWrongValue;
      JU    S128;	//-->Send 128
//==================================================
//Send Dataset 128
S128: L     128;
      T     #DPData.NrSndDataSet;
      L     0;
      T     #DPData.IdxSndDataSet;
      L     #InWeight;
      T     #DPData.Data.Value8;
      L     0;
      T     #DPData.Data.Value12;
      T     #DPData.Data.Value16;
      T     #DPData.Data.Value20;
      T     #DPData.Data.Value21;
      T     #DPData.Data.Value22;
      T     #DPData.Data.Value23;
      L     #InRecipeNr;
      T     #DPData.Data.Value21;
      JU    Snd;
//======================================================
//Send Dataset 136
S136: A     #Recipe.CmdSend;
      JCN   S000;
      L     136;
      T     #DPData.NrSndDataSet;
      L     #Recipe.InRecipeNr;
      T     #DPData.IdxSndDataSet;
      CALL  "SIEMENS_BLKMOV" (
           SRCBLK                   := #Recipe.Para,
           RET_VAL                  := #tmpReturn,
           DSTBLK                   := #DPData.Data);
      L     #Recipe.Para.InOutDosingSpeedFast;
      T     #DPData.Data.Value22;
      L     #Recipe.Para.InOutDosingSpeedSlow;
      T     #DPData.Data.Value23;
      JU    Snd;
//======================================================
//Send Dataset 0
S000: L     0;
      T     #DPData.NrSndDataSet;
      L     0;
      T     #DPData.IdxSndDataSet;
//======================================================
//Senden DP
Snd:  CALL  "SIEMENS_BLKMOV" (
           SRCBLK                   := #Par.Command,
           RET_VAL                  := #tmpReturn,
           DSTBLK                   := #DPData.StatusCommand);
      A     #InSimulation;
      JC    sSim;
      CALL  "SIEMENS_DPWR_DAT" (
           LADDR                    := #tmpAddr,
           RECORD                   := #DPData,
           RET_VAL                  := #tmpReturn);
      L     #tmpReturn;
      L     0;
      <>I;
      =     #Par.HelpFlags.OutComFaultSend;
      JU    sEnd;
//write to Simulation
sSim: R     #Par.HelpFlags.OutComFaultSend;
      A     "GCS7_Gr_SimDPtoImage";
      L     P#Q 0.0;
      JC    rDB2;
      OPN   "TEST_IOSimuliOutput";
      L     P#DBX 0.0;
rDB2: L     #Par.ParIOByteNr;
      SLD   3;
      +D;
      LAR1;
      L     #DPData.StatusCommand;
      T     D [AR1,P#0.0];
      L     #DPData.NrSndDataSet;
      T     B [AR1,P#4.0];
      L     #DPData.IdxSndDataSet;
      T     B [AR1,P#5.0];
      L     #DPData.NrRcvDataSet;
      T     B [AR1,P#6.0];
      L     #DPData.IdxRcvDataSet;
      T     B [AR1,P#7.0];
      L     #DPData.Data.Value8;
      T     D [AR1,P#8.0];
      L     #DPData.Data.Value12;
      T     D [AR1,P#12.0];
      L     #DPData.Data.Value16;
      T     D [AR1,P#16.0];
      L     #DPData.Data.Value20;
      T     B [AR1,P#20.0];
      L     #DPData.Data.Value21;
      T     B [AR1,P#21.0];
      L     #DPData.Data.Value22;
      T     B [AR1,P#22.0];
      L     #DPData.Data.Value23;
      T     B [AR1,P#23.0];
sEnd: NOP   0;
      NOP   0;
NETWORK
TITLE = State Code
//--Passive ---
      L     41;	//Code: Passive.HWStop
      A     #InHWStop;
      A     #StPassive;
      JC    STC;
      L     1;	//Code: Passive
      A     #StPassive;
      JC    STC;
      L     2;	//Code: starting
      A     #StStarting;
      JC    STC;
      L     3;	//Code: dosing
      A     #StDosing;
      JC    STC;
      L     14;	//Code: Suspended.Resulting
      A     #StSuspended;
      A     #Out_F_ResultIngr;
      JC    STC;
      L     44;	//Code: Suspended.HWStop
      A     #InHWStop;
      A     #StSuspended;
      JC    STC;
      L     4;	//Code: Suspended
      A     #StSuspended;
      JC    STC;
      L     5;	//Code: waiting
      A     #StWaiting;
      JC    STC;
      L     9;	//Code: emptying
      A     #StEmptying;
      JC    STC;
      L     10;	//Code: emptied
      A     #StEmptied;
      JC    STC;
      L     32;	//Code: fault
STC:  L     #StCode;	//Old state code
      TAK;
      T     #StCode;	//Save state code
      <>I;
      L     3;	//Load code for CBit methode
      CC    "SYS_CBitCtrl";
END_FUNCTION_BLOCK

FUNCTION_BLOCK "GCS7_M_Scourer"	// FB 44
TITLE = Scourer
//  
//COPYRIGHT:    (C) 1997  BUHLER AG, CH-9240 UZWIL, SWITZERLAND
//
//PRODUCT:      GCS7
//
//TITLE:        FB 44 Machine Control:Scourer 
//
//-------------------------------------------------------------------------
//
//IDENT:        AUTHOR:             DEPT:                       DATE:
//
//FB44.5.6      A. Egli             CT3                         30-Aug-2009
//              Manual mode if Bypassed
//FB44.5.5      K. Tischer          CT3                         13-Feb-2004
//              - StBypassed-->StStopping
//FB44.5.4      A. Egli             CT3                         24-Nov-2003
//              - Condition for Started
//FB44.5.3      A. Egli             CT3                         11-Nov-2003
//              - StStopping-->StBypassed
//              - StStarted -->StStopping
//FB44.5.2      A. Egli             CT3                         12-Sep-2003
//              No command Scourer.CmdNext as long InSeqStop
//FB44.5.1      A. Egli             CT3                         22-Jul-2003
//              Scourer.InLocal 
//FB44.5.0      A. Egli             CT3                         17-Jun-2002
//              New Release with one block 
//FB44.4.3      Ph. Engler          MU664                       03-Apr-2002
//              - Transition from stBypassed to stStarted
//                only if Flap.StHn
//              - Scourer.InLocal reset only if not Flap.StHn
//FB44.4.2      A. Egli             CT3                         24-Mai-2002
//              Set Scourer to local, if machine is bypassed
//FB44.4.1      Ph. Engler          MU664                       13-Mar-2002
//              - Screw: CmdFaultReset corrected
//              - Machine: stFault corrected
//              - Screw: InSeqStop if bypassed integrated
//FB44.4.0      A. Egli             CT3                         24-Mai-2000
//              Screw and Scraper 
//FB44.3.1      S.Kalberer          CT3                         10-Dec-1999
//              Scourer motor seqstops on Aspiration fan fault
//FB44.3.0      A. Egli             CT3                         11-Oct-1999
//              Local data reduced 
//FB44.2B       K. Tischer          MU664                       06-Mrz-1999
//              CC FC2 not UC FC2
//FB44.2A       A. Egli             CT3                         04-Mai-1998
//              StFault = StCode 32
//FB44.1A       A.Egli              AEE61                       12-Nov-1997
//              1st Release in S7
//
//-------------------------------------------------------------------------
//
//PURPOSE:      MANUAL : see [LL.MHXENMAN]
//
//RESTRICTIONS: S7
//              ACCU2: Pointer to dynamic datas of the machine
//              ACCU1: Pointer to parameter datas of the machine
//
//-------------------------------------------------------------------------
//
//
AUTHOR : EA
FAMILY : GCS7LL
NAME : Scourer
VERSION : 5.6
VAR
  Ma : UDT 20440;
  AspLow : FB 12;	//Element
  AspHigh : FB 12;	//Element
  Scourer : FB 12;	//Element
  ManFlap : FB 13;	//Element
  HL : FB 14;	//Element
  Screw : FB 12;	//Element
  Scraper : FB 11;	//Element
END_VAR
VAR_TEMP
  tmpFaultStop : BOOL ;
  tmpFaultSum : BOOL ;
  tmpStopped : BOOL ;
  tmpOffsetInstanzDB : DWORD ;
  tmpAddrParMa : DWORD ;	//Byte Nr of first Parameter in Instanz DB
  tmpAddrParaElement : DWORD ;
  tmpNext : BOOL ;
  tmpLocal : BOOL ;
  tmpEnable : BOOL ;
  tmpEnableOpen : BOOL ;
  tmpEmpty : BOOL ;
  tmpLenDyn : INT ;
  tmpStarted : BOOL ;	//all elemenet started , without Scourer
  StoreGrOutManualOff : BOOL ;
END_VAR
BEGIN
NETWORK
TITLE =
      L     10;
      T     #tmpLenDyn;
NETWORK
TITLE = PC Control
//=== Test Object number =====================
      L     "SYS_DirectCtrlDB".PC.ObjectNo;	//PCControl.ObjectNo
      L     #Ma.Par.ParObjectNo;	//Input ObjectNo
      <>I;
      JC    aEnd;
//=== Test OType      ========================
      L     2044;	//Input object type
      L     "SYS_DirectCtrlDB".PC.ObjectType;	//PCControl.ObjectType
      <>I;
      JC    aEnd;
//=== Test Handshake =========================
      A     "SYS_DirectCtrlDB".PC.Hsk.FExamine;	// Handshake.FExamine
      JC    aExa;
      A     "SYS_DirectCtrlDB".PC.Hsk.FDefineCmd;	// Handshake.FDefineCmd
      O     "SYS_DirectCtrlDB".PC.Hsk.FDefinePara;	// Handshake.FDefinePara
      JC    aCmd;
aIni: L     2;	// FcInit
      UC    "SYS_DirectCtrl";
      JU    aEnd;
// Write new commands from PC to Interface of group 
aCmd: A     "SYS_DirectCtrlDB".PC.Cmd1[8];	//Cmd1[8]=CmdOff
      S     #Ma.CmdOff;
      A     "SYS_DirectCtrlDB".PC.Cmd1[9];	//Cmd1[9]=CmdOn
      S     #Ma.CmdOn;
      A     "SYS_DirectCtrlDB".PC.Cmd1[10];	//Cmd1[10]=CmdNext
      S     #Ma.CmdNext;
      A     "SYS_DirectCtrlDB".PC.Cmd1[11];	//Cmd1[11]=CmdFaultReset
      S     #Ma.CmdFaultReset;
      A     "SYS_DirectCtrlDB".PC.Cmd1[13];	//Cmd1[13]=CmdManualOn
      S     #Ma.InManual;
      A     "SYS_DirectCtrlDB".PC.Cmd2[13];	//Cmd1[13]=CmdManualOff
      R     #Ma.InManual;
      AN    "SYS_DirectCtrlDB".PC.Hsk.FDefinePara;	// Handshake.FDefinePara
      JC    aIni;
      JU    aIni;
aExa: TAR2;	// Address Dynamic data
      T     "SYS_DirectCtrlDB".GC.InDynAddr;	// -->PCControl.GC.InDynAddr
      L     #tmpLenDyn;	// Length Dynamic data
      T     "SYS_DirectCtrlDB".GC.InDynLen;	// -->PCControl.GC.InDynLen
      L     0;
      T     "SYS_DirectCtrlDB".GC.InParaAddr;	// -->PCControl.GC.InParaAddr
      T     "SYS_DirectCtrlDB".GC.InParaLen;	// -->PCControl.GC.InParaLen
      L     1;	// Code FcExamine
      UC    "SYS_DirectCtrl";
      L     10;	//Revision
      T     "SYS_DirectCtrlDB".GC.Revision;
aEnd: NOP   0;
NETWORK
TITLE = Interlocking
//===Global Group Orders===
      A     "GCS7_Gr_OutManualOn";	//Gr.OutManualOn
      S     #Ma.InManual;
      A     "GCS7_Gr_OutManualOff";	//Gr.OutManualOff
      R     #Ma.InManual;
      A     #Ma.InManual;
      S     "GCS7_Gr_InManual";	//Gr.InManual
      A     #Ma.CmdNext;
      AN    #Ma.InManual;
      O     #Ma.CmdOn;
      =     #tmpNext;
      A     #Ma.InLocal;
      AN    #Ma.InManual;
      =     #tmpLocal;
      AN    #tmpLocal;
      A     #Ma.InEnable;
      AN    #Ma.CmdOff;
      =     #tmpEnable;
//--- Fault----
      A     #AspLow.StFault;
      O     #AspHigh.StFault;
      O;
      A     #Scourer.StFault;	// [5.6]
      AN    #ManFlap.StHN;	// [5.6]
      O     #HL.StFault;
      O     #ManFlap.StFault;
      O     #Screw.StFault;	// [4.1]
      O     #Scraper.StFault;	// [4.1]
      =     #tmpFaultSum;
//--- Next
      AN    #Ma.Par.ParWithScrew;
      JC    InX1;
      A     #tmpNext;
      S     #Screw.CmdNext;
InX1: AN    #Ma.Par.ParWithScraper;
      JC    InX2;
      A     #tmpNext;
      S     #Scraper.CmdNext;
InX2: A(;
      O     #Screw.StStartedFwd;
      ON    #Ma.Par.ParWithScrew;
      );
      A(;
      O     #Scraper.StStarted;
      ON    #Ma.Par.ParWithScraper;
      );
      A     #tmpNext;
      S     #AspLow.CmdNext;
      A     #AspLow.StStartedFwd;
      A     #tmpNext;
      S     #AspHigh.CmdNext;
      A     #AspHigh.StStartedFwd;	// 3.1:
      ON    #Ma.Par.ParWithAspHigh;	// 3.1:
      A     #AspLow.StStartedFwd;	// 3.1:
      A     #tmpNext;	// 3.1:
      AN    #Scourer.InSeqStop;	//[5.2]
      S     #Scourer.CmdNext;
//--- Interlocking
      AN    #Ma.Par.ParWithScrew;
      JC    InE1;
      A     #tmpEnable;
      =     #Screw.InEnableFwd;
InE1: AN    #Ma.Par.ParWithScraper;
      JC    InE2;
      A(;
      O     #Screw.StStartedFwd;
      ON    #Ma.Par.ParWithScrew;
      );
      A     #tmpEnable;
      =     #Scraper.InEnable;
InE2: A     #tmpEnable;
      =     #AspLow.InEnableFwd;
      A     #tmpEnable;
      =     #AspHigh.InEnableFwd;
      A(;
      A     #Screw.StStartedFwd;
      ON    #Ma.Par.ParWithScrew;
      );
      A(;
      A     #Scraper.StStarted;
      ON    #Ma.Par.ParWithScraper;
      );
      A     #tmpEnable;
//      UN    #ManFlap.StHN // [4.1]
      =     #Scourer.InEnableFwd;
//Sequenz stop
      AN    #Ma.InManual;
      A     #Ma.InSeqStop;
      =     #AspLow.InSeqStop;
      =     #AspHigh.InSeqStop;
      AN    #Ma.Par.ParWithScrew;
      JC    InQ1;
      A     #AspLow.InSeqStop;
      =     #Screw.InSeqStop;
InQ1: AN    #Ma.Par.ParWithScraper;
      JC    InQ2;
      A     #AspLow.InSeqStop;
      =     #Scraper.InSeqStop;
InQ2: A     #AspHigh.StFault;	// 3.1:
      A     #Ma.Par.ParWithAspHigh;	// 3.1:
      O     #AspLow.StFault;	// 3.1:
      O     #AspLow.InSeqStop;
      O     #ManFlap.StHN;	// [4.1]
      =     #Scourer.InSeqStop;
//--- Local mode --
      A     #tmpLocal;
      =     #AspLow.InLocal;
      =     #AspHigh.InLocal;
      =     #ManFlap.InLocal;
      =     #HL.InLocal;
      AN    #tmpLocal;	// [4.2]
      AN    #ManFlap.StHN;	// [4.3]
      R     #Scourer.InLocal;	// [4.2]
      A     #ManFlap.StHN;	// [4.2]
      A     #Scourer.StStopped;	// [4.2]
      O     #tmpLocal;	// [5.1]
      S     #Scourer.InLocal;	// [4.2]
      AN    #Ma.Par.ParWithScrew;
      JC    InL1;
      A     #tmpLocal;
      =     #Screw.InLocal;
InL1: AN    #Ma.Par.ParWithScraper;
      JC    InL2;
      A     #tmpLocal;
      =     #Scraper.InLocal;
//--- Fault Reset -------------
InL2: A     #Ma.CmdFaultReset;
      S     #AspLow.CmdFaultReset;
      S     #AspHigh.CmdFaultReset;
      S     #Scourer.CmdFaultReset;
      S     #ManFlap.CmdFaultReset;
      S     #HL.CmdFaultReset;
      AN    #Ma.Par.ParWithScrew;
      JC    InF1;
      A     #Ma.CmdFaultReset;	// [4.1]
      S     #Screw.CmdFaultReset;
InF1: AN    #Ma.Par.ParWithScraper;
      JC    InF2;
      A     #Ma.CmdFaultReset;
      S     #Scraper.CmdFaultReset;
//--- Monitoring HL
InF2: SET;
      S     #HL.InMonFalse;
NETWORK
TITLE = Call AspLow
      CALL  #AspLow;
NETWORK
TITLE = Call AspHigh
      AN    #Ma.Par.ParWithAspHigh;
      JC    el3;
      CALL  #AspHigh;
NETWORK
TITLE = Call Scourer
el3:  A     "GCS7_Gr_OutManualOff";	//[5.6]
      =     #StoreGrOutManualOff;	//[5.6]
      A     #ManFlap.StHN;	//[5.6]
      AN    #Ma.InLocal;	//[5.6]
      R     "GCS7_Gr_OutManualOff";	//[5.6]
      CALL  #Scourer;
      A     #StoreGrOutManualOff;	//[5.6]
      =     "GCS7_Gr_OutManualOff";	//[5.6]
NETWORK
TITLE = Call ManFlap
      CALL  #ManFlap;
NETWORK
TITLE = Call Digital Input: HL
      AN    #Ma.Par.ParWithHL;
      JC    HLen;
      CALL  #HL;
HLen: NOP   0;
NETWORK
TITLE = Call Motor: Screw
      AN    #Ma.Par.ParWithScrew;
      JC    SCen;
      CALL  #Screw;
SCen: NOP   0;
NETWORK
TITLE = Call Digital Output: Scraper
      AN    #Ma.Par.ParWithScraper;
      JC    SPen;
      CALL  #Scraper;
SPen: NOP   0;
NETWORK
TITLE = Jump to actual state
      A     #AspHigh.StStopped;
      ON    #Ma.Par.ParWithAspHigh;
      A     #AspLow.StStopped;
      A     #Scourer.StStopped;
      A(;
      A     #Screw.StStopped;
      ON    #Ma.Par.ParWithScrew;
      );
      A(;
      A     #Scraper.StStopped;
      ON    #Ma.Par.ParWithScraper;
      );
      =     #tmpStopped;
//[5.3]--->
      A     #AspHigh.StStartedFwd;
      ON    #Ma.Par.ParWithAspHigh;
      A     #AspLow.StStartedFwd;
      A(;
      A     #Screw.StStartedFwd;
      ON    #Ma.Par.ParWithScrew;
      );
      A(;
      A     #Scraper.StStarted;
      ON    #Ma.Par.ParWithScraper;
      );
      A(;	//[5.4]
      A     #Scourer.StStartedFwd;	//[5.4]
      O     #ManFlap.StHN;	//[5.4]
      O     #ManFlap.StCtoLN;	//[5.4]
      );	//[5.4]
      =     #tmpStarted;
// <---[5.3]
//====================================
      A     #Ma.StStopped;
      JC    S0;	// ===> State
      A     #Ma.StStarted;
      JC    S2;	// ===> State
      A     #Ma.StStarting;
      JC    S1;	// ===> State
      A     #Ma.StStopping;
      JC    S3;	// ===> State
      A     #Ma.StFault;
      JC    S4;	// ===> State
      A     #Ma.StBypassed;
      JC    S6;	// ===> State
NETWORK
TITLE = Stopped
//any Transition 
xxS0: S     #Ma.StStopped;	// ===> Initialisation
//=== Logic
// Condition for StFault
S0:   A     #tmpFaultSum;
      R     #Ma.StStopped;
      JC    xxS4;	//--> ST_FAULT:
// Condition for StStarting
      AN    #tmpStopped;
      R     #Ma.StStopped;
      JC    xxS1;	//--> StStarting
      JU    OUT;
NETWORK
TITLE = StStarting
//any Transition 
xxS1: S     #Ma.StStarting;
//=== Logic
// Condition for StFault
S1:   A     #tmpFaultSum;
      R     #Ma.StStarting;
      JC    xxS4;	//--> StFault
// Condition for StStarted
      A     #tmpStarted;	//[5.3]
      A     #Scourer.StStartedFwd;
      R     #Ma.StStarting;
      JC    xxS2;	//-->StStarted
// Condition for StBypassed
      A     #tmpStarted;	//[5.3]
      A     #ManFlap.StHN;
      R     #Ma.StStarting;
      JC    xxS6;	//-->StBypassed
// Condition for StStopping
      A     #AspLow.InSeqStop;
      ON    #AspLow.InEnableFwd;
      O     #tmpStopped;
      R     #Ma.StStarting;
      JC    xxS3;	//-->StStopping
      JU    OUT;
NETWORK
TITLE = StStarted
//any Transition 
xxS2: S     #Ma.StStarted;
//=== Logic
// Condition for StFault
S2:   A     #tmpFaultSum;
      R     #Ma.StStarted;
      JC    xxS4;	//--> StFault
// Condition for StBypassed
      A     #tmpStarted;	//[5.3]
      A     #ManFlap.StHN;
      R     #Ma.StStarted;
      JC    xxS6;	//-->StBypassed
// Condition for StStopping
      AN    #tmpStarted;	//[5.3]
      ON    #Scourer.StStartedFwd;
      R     #Ma.StStarted;
      JC    xxS3;	//-->StStopping
      JU    OUT;
NETWORK
TITLE = Stopping
//any Transition 
xxS3: S     #Ma.StStopping;
      JU    OUT;	//[5.4]
//=== Logic
// Condition for StFault
S3:   A     #tmpFaultSum;
      R     #Ma.StStopping;
      JC    xxS4;	//--> StFault
// Condition for StStopped
      A     #tmpStopped;
      R     #Ma.StStopping;
      JC    xxS0;	//-->StStopped
// Condition for StStarting
      A     #tmpStarted;	//[5.3]
      AN    #ManFlap.StHN;
      R     #Ma.StStopping;
      JC    xxS1;	//-->StStarting
// Condition for StBypassed             //[5.3]
      A     #tmpStarted;	//[5.3]
      A     #ManFlap.StHN;	//[5.3]
      R     #Ma.StStopping;	//[5.3]
      JC    xxS6;	//[5.3]-->StBypassed 
      JU    OUT;
NETWORK
TITLE = Fault
//any Transition 
xxS4: S     #Ma.StFault;
//=== Logic
S4:   A     #tmpFaultSum;
      JC    OUT;
//---- Transition --
      R     #Ma.StFault;
      JU    xxS1;	//-->StStopping 
NETWORK
TITLE = StBypassed
//any Transition 
xxS6: S     #Ma.StBypassed;
//=== Logic
// Condition for StFault
S6:   A     #tmpFaultSum;
      R     #Ma.StBypassed;
      JC    xxS4;	//--> StFault
// Condition for StStarted
      A     #tmpStarted;	//[5.3]
      A     #Scourer.StStartedFwd;
      A     #ManFlap.StLN;	// [4.3]
      R     #Ma.StBypassed;
      JC    xxS2;	//-->StStarted
// Condition for StStopping
      A     #Scourer.StStopped;
      AN    #ManFlap.StHN;
      AN    #ManFlap.StCtoLN;
      ON    #tmpStarted;	//[5.3]
      AN    #Scourer.StStarting;	//[5.5]
      R     #Ma.StBypassed;
      JC    xxS3;	//-->StStopping
      JU    OUT;
NETWORK
TITLE = State Code
// State     StCode
// ----------------------
// StFault32
// StStopped    1
// StStarting   2
// StStarted.Wait   3
// StStarted.Feeding4
// StEmptying    5
// StBypassed    6
// StStopping  7
OUT:  A     #Ma.StStopped;
      L     1;	//Code=StStopped
      JC    Code;
      A     #Ma.StStarted;
      L     3;	//Code=StStarted
      JC    Code;
      A     #Ma.StBypassed;
      L     9;	//Code=StBypassed
      JC    Code;
      A     #Ma.StStarting;
      L     2;	//Code=StStarting
      JC    Code;
      A     #Ma.StStopping;
      L     7;	//Code=StStopping 
      JC    Code;
      L     32;	//Code=StFault 
Code: L     #Ma.StCode;	// Old state code
      TAK;
      T     #Ma.StCode;	// Save state code
      <>I;
      L     3;
      CC    "SYS_CBitCtrl";	//Set change bit
NETWORK
TITLE = Global End
      CLR;	//---Clear all commands
      =     #Ma.CmdOn;
      =     #Ma.CmdOff;
      =     #Ma.CmdNext;
      =     #Ma.CmdFaultReset;
END_FUNCTION_BLOCK

FUNCTION_BLOCK "GCS7_M_Roll4Stand"	// FB 45
TITLE = 4 roll stand
//  
//COPYRIGHT:    (C) 1997  BUHLER AG, CH-9240 UZWIL, SWITZERLAND
//
//PRODUCT:      GCS7
//
//TITLE:        FB 45 Machine 4 roll stand
//
//-------------------------------------------------------------------------
//
//IDENT:        AUTHOR:             DEPT:                       DATE:
//
//FB45.4.2      A. Egli             CT3                         05-Mai-2004
//              CmdOff in manual mode
//FB45.4.1      A. Egli             CT3                         23-Sep-2003
//              InEnable=0 must stop motor when ParManual=1 and InManual=0
//FB45.4.0      A. Egli             CT3                         17-Jun-2002
//              New Release with one block 
//FB45.3.1      A. Egli             CT3                         08-Feb-2000
//              Condition Monitoring HL 
//FB45.3.0      A. Egli             CT3                         11-Oct-1999
//              Local data reduced 
//FB45.2B       K. Tischer          MU664                       06-Mrz-1999
//              CC FC2 not UC FC2
//FB45.2A       A. Egli             CT3                         04-Mai-1998
//              StFault = StCode 32
//FB45.1A       A.Egli              AEE61                       12-Nov-1997
//              1st Release in S7
//
//-------------------------------------------------------------------------
//
//PURPOSE:      MANUAL : see [LL.RL8xxMAN]
//
//RESTRICTIONS: S7
//              ACCU2: Pointer to dynamic datas of the machine
//              ACCU1: Pointer to parameter datas of the machine
//
//-------------------------------------------------------------------------
//
//
AUTHOR : EA
FAMILY : GCS7LL
NAME : Roll4
VERSION : 4.2
VAR
  Ma : UDT 20450;
  RollsLeft : FB 12;	//Element
  RollsRight : FB 12;	//Element
  SMLeft : FB 14;	//Element
  SMRight : FB 14;	//Element
  HLInletLeft : FB 14;	//Element
  HLInletRight : FB 14;	//Element
END_VAR
VAR_TEMP
  tmpFaultSum : BOOL ;
  tmpWarning : BOOL ;
  tmpStarted : BOOL ;
  tmpNext : BOOL ;
  tmpLocal : BOOL ;
  tmpEnable : BOOL ;
  tmpSeqStop : BOOL ;
  tmpLenDyn : INT ;
END_VAR
BEGIN
NETWORK
TITLE =
      L     10;
      T     #tmpLenDyn;
NETWORK
TITLE = PC Control
//=== Test Object number =====================
      L     "SYS_DirectCtrlDB".PC.ObjectNo;	//PCControl.ObjectNo
      L     #Ma.Par.ParObjectNo;	//Input ObjectNo    
      <>I;
      JC    aEnd;
//=== Test OType      ========================
      L     2045;	//Input object type
      L     "SYS_DirectCtrlDB".PC.ObjectType;	//PCControl.ObjectType
      <>I;
      JC    aEnd;
//=== Test Handshake =========================
      A     "SYS_DirectCtrlDB".PC.Hsk.FExamine;	// Handshake.FExamine
      JC    aExa;
      A     "SYS_DirectCtrlDB".PC.Hsk.FDefineCmd;	// Handshake.FDefineCmd
      O     "SYS_DirectCtrlDB".PC.Hsk.FDefinePara;	// Handshake.FDefinePara
      JC    aCmd;
aIni: L     2;	// FcInit
      UC    "SYS_DirectCtrl";
      JU    aEnd;
// Write new commands from PC to Interface of group 
aCmd: A     "SYS_DirectCtrlDB".PC.Cmd1[1];	//Cmd1[1]=CmdEnableLeft
      R     #Ma.InDisableLeft;
      A     "SYS_DirectCtrlDB".PC.Cmd2[1];	//Cmd2[1]=CmdDisableLeft
      S     #Ma.InDisableLeft;
      A     "SYS_DirectCtrlDB".PC.Cmd1[2];	//Cmd1[2]=CmdEnableRight
      R     #Ma.InDisableRight;
      A     "SYS_DirectCtrlDB".PC.Cmd2[2];	//Cmd2[2]=CmdDisableRight
      S     #Ma.InDisableRight;
      A     "SYS_DirectCtrlDB".PC.Cmd1[3];	//Cmd1[3]=CmdOverwriteHLOn
      S     #Ma.InOverrideHL;
      A     "SYS_DirectCtrlDB".PC.Cmd2[3];	//Cmd2[3]=CmdOverwriteHLOff
      R     #Ma.InOverrideHL;
      A     "SYS_DirectCtrlDB".PC.Cmd1[8];	//Cmd1[8]=CmdOff
      S     #Ma.CmdOff;
      A     "SYS_DirectCtrlDB".PC.Cmd1[9];	//Cmd1[9]=CmdOn
      S     #Ma.CmdOn;
      A     "SYS_DirectCtrlDB".PC.Cmd1[10];	//Cmd1[10]=CmdNext
      S     #Ma.CmdNext;
      A     "SYS_DirectCtrlDB".PC.Cmd1[11];	//Cmd1[11]=CmdFaultReset
      S     #Ma.CmdFaultReset;
      A     "SYS_DirectCtrlDB".PC.Cmd1[13];	//Cmd1[13]=CmdManualOn
      S     #Ma.InManual;
      A     "SYS_DirectCtrlDB".PC.Cmd2[13];	//Cmd1[13]=CmdManualOff
      R     #Ma.InManual;
      AN    "SYS_DirectCtrlDB".PC.Hsk.FDefinePara;	// Handshake.FDefinePara
      JC    aIni;
      JU    aIni;
aExa: TAR2;	// Address Dynamic data
      T     "SYS_DirectCtrlDB".GC.InDynAddr;	// -->PCControl.GC.InDynAddr
      L     #tmpLenDyn;	// Length Dynamic data
      T     "SYS_DirectCtrlDB".GC.InDynLen;	// -->PCControl.GC.InDynLen
      L     0;
      T     "SYS_DirectCtrlDB".GC.InParaAddr;	// -->PCControl.GC.InParaAddr
      T     "SYS_DirectCtrlDB".GC.InParaLen;	// -->PCControl.GC.InParaLen
      L     1;	// Code FcExamine
      UC    "SYS_DirectCtrl";
      L     10;	//Revision
      T     "SYS_DirectCtrlDB".GC.Revision;
aEnd: NOP   0;
NETWORK
TITLE = Interlocking
//===Global Group Orders===
      A     "GCS7_Gr_OutManualOn";	//Gr.OutManualOn
      S     #Ma.InManual;
      A     "GCS7_Gr_OutManualOff";	//Gr.OutManualOff
      R     #Ma.InManual;
      A     #Ma.InManual;
      S     "GCS7_Gr_InManual";	//Gr.InManual
// temporare
      AN    #Ma.StStarting;
      ON    #Ma.InManual;
      O     #Ma.CmdOff;	//[4.2]
      R     #Ma.OutStartMan;
      O     #Ma.CmdOn;
      S     #Ma.OutStartMan;
      A     #Ma.CmdNext;
      AN    #Ma.InManual;
      O     #Ma.OutStartMan;
      =     #tmpNext;
      A     #Ma.InManual;
      ON    #Ma.InLocal;
      A(;
      A     #Ma.Par.ParManual;	//[4.1]
      A     #Ma.InManual;
      O     #Ma.InEnable;
      );
      AN    #Ma.CmdOff;
      =     #tmpEnable;
      A     #Ma.InSeqStop;
      AN    #Ma.InManual;
      =     #tmpSeqStop;
//--- Fault----
      A     #RollsLeft.StFault;
      O     #RollsRight.StFault;
      =     #tmpWarning;
      A     #tmpWarning;
      AN    #Ma.Par.ParWarning;
      O     #HLInletLeft.StFault;
      O     #SMLeft.StFault;
      O     #HLInletRight.StFault;
      O     #SMRight.StFault;
      =     #tmpFaultSum;
//--- Next
      A     #tmpNext;
      S     #RollsLeft.CmdNext;
      A     #RollsLeft.StStartedFwd;
      O     #Ma.InDisableLeft;
      A     #tmpNext;
      S     #RollsRight.CmdNext;
//--- Interlocking Motors
//RollLeft
      A     #tmpEnable;
      AN    #Ma.InDisableLeft;
      =     #RollsLeft.InEnableFwd;
// 
      A     #tmpSeqStop;
      =     #RollsLeft.InSeqStop;
//RollRight
      A     #tmpEnable;
      AN    #Ma.InDisableRight;
      =     #RollsRight.InEnableFwd;
// 
      A     #tmpSeqStop;
      =     #RollsRight.InSeqStop;
// 
//--- Local mode --
      A     #Ma.InLocal;
      AN    #Ma.InManual;
      =     #RollsLeft.InLocal;
      =     #SMLeft.InLocal;
      =     #RollsRight.InLocal;
      =     #SMRight.InLocal;
      =     #HLInletLeft.InLocal;
      =     #HLInletRight.InLocal;
//--- Fault Reset -------------
      A     #Ma.CmdFaultReset;
      S     #RollsLeft.CmdFaultReset;
      S     #HLInletLeft.CmdFaultReset;
      S     #SMLeft.CmdFaultReset;
      S     #RollsRight.CmdFaultReset;
      S     #HLInletRight.CmdFaultReset;
      S     #SMRight.CmdFaultReset;
// 
//--- Monitoring 
      AN    #Ma.InOverrideHL;	//[3.1] 
      =     #HLInletLeft.InMonFalse;	//[3.1] 
      =     #HLInletRight.InMonFalse;	//[3.1] 
      A     #Ma.InpPressureLeft;
      =     #SMLeft.InMonTrue;
      A     #Ma.InpPressureRight;
      =     #SMRight.InMonTrue;
//Startup done
      A     #RollsLeft.StStartedFwd;
      O     #RollsLeft.StFault;
      O     #Ma.InDisableLeft;
      A(;
      O     #RollsRight.StStartedFwd;
      O     #RollsRight.StFault;
      O     #Ma.InDisableRight;
      );
      =     #Ma.OutStartupDone;
      A     #RollsLeft.StStartedFwd;
      O     #Ma.InDisableLeft;
      A(;
      O     #RollsRight.StStartedFwd;
      O     #Ma.InDisableRight;
      );
      A(;
      ON    #Ma.InDisableLeft;
      ON    #Ma.InDisableRight;
      );
      =     #tmpStarted;
NETWORK
TITLE = Call RollLeft
      CALL  #RollsLeft;
NETWORK
TITLE = Call Digital Input: HLInletLeft
      AN    #Ma.Par.ParWithHLInletLeft;
      JC    elL5;
      CALL  #HLInletLeft;
NETWORK
TITLE = Call Digital Input: SMLeft
elL5: AN    #Ma.Par.ParWithSMLeft;
      JC    elL7;
      CALL  #SMLeft;
NETWORK
TITLE = Call RollRight
elL7: CALL  #RollsRight;
NETWORK
TITLE = Call Digital Input: HLInletRight
      AN    #Ma.Par.ParWithHLInletRight;
      JC    elR5;
      CALL  #HLInletRight;
NETWORK
TITLE = Call Digital Input: SMRight
elR5: AN    #Ma.Par.ParWithSMRight;
      JC    StJ0;
      CALL  #SMRight;
NETWORK
TITLE = Actual State
// StFault
StJ0: A     #tmpFaultSum;
      =     #Ma.StFault;
// StWarning
      A     #tmpWarning;
      A     #Ma.Par.ParWarning;
      AN    #Ma.StFault;
      =     #Ma.StWarning;
// StStopped
      A     #RollsLeft.StStopped;
      A     #RollsRight.StStopped;
      AN    #Ma.StFault;
      =     #Ma.StStopped;
// StStarted
      A     #tmpStarted;
      AN    #Ma.StFault;
      AN    #Ma.StStopped;
      =     #Ma.StStarted;
// StStopping
      A     #RollsLeft.InSeqStop;
      O     #RollsRight.InSeqStop;
      AN    #Ma.StStarted;
      AN    #Ma.StStopped;
      AN    #Ma.StFault;
      AN    #Ma.StWarning;
      =     #Ma.StStopping;
// StStarting
      AN    #Ma.StStopped;
      AN    #Ma.StStarted;
      AN    #Ma.StStopping;
      AN    #Ma.StFault;
      AN    #Ma.StWarning;
      =     #Ma.StStarting;
NETWORK
TITLE = State Code
// State     StCode
// ----------------------
// StFault32
// StStopped    1
// StStarting   2
// StStarted   3
// StStopping  7
// StWarning8
      A     #Ma.StStopped;
      L     1;	//Code=StStopped
      JC    Code;
      A     #Ma.StStarted;
      L     3;	//Code=StStarted
      JC    Code;
      A     #Ma.StWarning;
      L     8;	//Code=StWarning 
      JC    Code;
      A     #Ma.StStarting;
      L     2;	//Code=StStarting
      JC    Code;
      A     #Ma.StStopping;
      L     7;	//Code=StStopping 
      JC    Code;
      L     32;	//Code=StFault 
Code: L     #Ma.StCode;	// Old state code
      TAK;
      T     #Ma.StCode;	// Save state code
      <>I;
      L     3;
      CC    "SYS_CBitCtrl";	//Set change bit
NETWORK
TITLE = Global End
      CLR;	//---Clear all commands
      =     #Ma.CmdOn;
      =     #Ma.CmdOff;
      =     #Ma.CmdNext;
      =     #Ma.CmdFaultReset;
END_FUNCTION_BLOCK

FUNCTION_BLOCK "GCS7_M_Roll8Stand"	// FB 46
TITLE = Roll stand with 8
//  
//COPYRIGHT:    (C) 1997  BUHLER AG, CH-9240 UZWIL,  SWITZERLAND
//
//PRODUCT:      GCS7
//
//TITLE:        FB 46 Machine roll stand with 8 rolls
//
//-------------------------------------------------------------------------
//
//IDENT:        AUTHOR:             DEPT:                       DATE:
//
//FB46.4.2      A. Egli             CT3                         05-Mai-2004
//              CmdOff in manual mode
//FB46.4.1      A. Egli             CT3                         23-Sep-2003
//              InEnable=0 must stop motor when ParManual=1 and InManual=0
//FB46.4.0      A. Egli             CT3                         18-Oct-2002
//              New Release with one block 
//FB46.3.2      A. Egli             CT3                         18-Okt-2002
//              Condition tmpStarted with ParMa.Par4Rolls=0 
//FB46.3.1      A. Egli             CT3                         08-Feb-2000
//              Condition Monitoring HL 
//FB46.3.0      A. Egli             CT3                         11-Oct-1999
//              Local data reduced 
//FB46.2B       K. Tischer          MU664                       06-Mrz-1999
//              CC FC2 not UC FC2
//FB46.2A       A. Egli             CT3                         04-Mai-1998
//              StFault = StCode 32
//FB46.1A       A.Egli              AEE61                       12-Nov-1997
//              1st Release in S7
//
//-------------------------------------------------------------------------
//
//PURPOSE:      MANUAL : see [LL.RL8xxMAN]
//
//RESTRICTIONS: S7
//              ACCU2: Pointer to dynamic datas of the machine
//              ACCU1: Pointer to parameter datas of the machine
//
//-------------------------------------------------------------------------
//
//
AUTHOR : EA
FAMILY : GCS7LL
NAME : Rolls8
VERSION : 4.2
VAR
  Ma : UDT 20460;
  RollsLowLeft : FB 12;	//Element
  RollsLowRight : FB 12;	//Element
  SpeedLeft : FB 14;	//Element
  SpeedRight : FB 14;	//Element
  HLInletLeft : FB 14;	//Element
  HLInletRight : FB 14;	//Element
  HLMidLeft : FB 14;	//Element
  HLMidRight : FB 14;	//Element
  RollsUpLeft : FB 12;	//Element
  RollsUpRight : FB 12;	//Element
END_VAR
VAR_TEMP
  tmpFaultSum : BOOL ;
  tmpWarning : BOOL ;
  tmpStarted : BOOL ;
  tmpNext : BOOL ;
  tmpLocal : BOOL ;
  tmpEnable : BOOL ;
  tmpSeqStop : BOOL ;
  tmpLenDyn : INT ;
END_VAR
BEGIN
NETWORK
TITLE =
      L     10;
      T     #tmpLenDyn;
NETWORK
TITLE = PC Control
//=== Test Object number =====================
      L     "SYS_DirectCtrlDB".PC.ObjectNo;	//PCControl.ObjectNo
      L     #Ma.Par.ParObjectNo;	//Input ObjectNo    
      <>I;
      JC    aEnd;
//=== Test OType      ========================
      L     2046;	//Input object type
      L     "SYS_DirectCtrlDB".PC.ObjectType;	//PCControl.ObjectType
      <>I;
      JC    aEnd;
//=== Test Handshake =========================
      A     "SYS_DirectCtrlDB".PC.Hsk.FExamine;	// Handshake.FExamine
      JC    aExa;
      A     "SYS_DirectCtrlDB".PC.Hsk.FDefineCmd;	// Handshake.FDefineCmd
      O     "SYS_DirectCtrlDB".PC.Hsk.FDefinePara;	// Handshake.FDefinePara
      JC    aCmd;
aIni: L     2;	// FcInit
      UC    "SYS_DirectCtrl";
      JU    aEnd;
// Write new commands from PC to Interface of group 
aCmd: A     "SYS_DirectCtrlDB".PC.Cmd1[1];	//Cmd1[1]=CmdEnableLeft
      R     #Ma.InDisableLeft;
      A     "SYS_DirectCtrlDB".PC.Cmd2[1];	//Cmd2[1]=CmdDisableLeft
      S     #Ma.InDisableLeft;
      A     "SYS_DirectCtrlDB".PC.Cmd1[2];	//Cmd1[2]=CmdEnableRight
      R     #Ma.InDisableRight;
      A     "SYS_DirectCtrlDB".PC.Cmd2[2];	//Cmd2[2]=CmdDisableRight
      S     #Ma.InDisableRight;
      A     "SYS_DirectCtrlDB".PC.Cmd1[3];	//Cmd1[3]=CmdOverwriteHLOn
      S     #Ma.InOverwriteHL;
      A     "SYS_DirectCtrlDB".PC.Cmd2[3];	//Cmd2[3]=CmdOverwriteHLOff
      R     #Ma.InOverwriteHL;
      A     "SYS_DirectCtrlDB".PC.Cmd1[8];	//Cmd1[8]=CmdOff
      S     #Ma.CmdOff;
      A     "SYS_DirectCtrlDB".PC.Cmd1[9];	//Cmd1[9]=CmdOn
      S     #Ma.CmdOn;
      A     "SYS_DirectCtrlDB".PC.Cmd1[10];	//Cmd1[10]=CmdNext
      S     #Ma.CmdNext;
      A     "SYS_DirectCtrlDB".PC.Cmd1[11];	//Cmd1[11]=CmdFaultReset
      S     #Ma.CmdFaultReset;
      A     "SYS_DirectCtrlDB".PC.Cmd1[13];	//Cmd1[13]=CmdManualOn
      S     #Ma.InManual;
      A     "SYS_DirectCtrlDB".PC.Cmd2[13];	//Cmd1[13]=CmdManualOff
      R     #Ma.InManual;
      AN    "SYS_DirectCtrlDB".PC.Hsk.FDefinePara;	// Handshake.FDefinePara
      JC    aIni;
      JU    aIni;
aExa: TAR2;	// Address Dynamic data
      T     "SYS_DirectCtrlDB".GC.InDynAddr;	// -->PCControl.GC.InDynAddr
      L     #tmpLenDyn;	// Length Dynamic data
      T     "SYS_DirectCtrlDB".GC.InDynLen;	// -->PCControl.GC.InDynLen
      L     0;
      T     "SYS_DirectCtrlDB".GC.InParaAddr;	// -->PCControl.GC.InParaAddr
      T     "SYS_DirectCtrlDB".GC.InParaLen;	// -->PCControl.GC.InParaLen
      L     1;	// Code FcExamine
      UC    "SYS_DirectCtrl";
      L     10;	//Revision
      T     "SYS_DirectCtrlDB".GC.Revision;
aEnd: NOP   0;
NETWORK
TITLE = Interlocking
//===Global Group Orders===
      A     "GCS7_Gr_OutManualOn";	//Gr.OutManualOn
      S     #Ma.InManual;
      A     "GCS7_Gr_OutManualOff";	//Gr.OutManualOff
      R     #Ma.InManual;
      A     #Ma.InManual;
      S     "GCS7_Gr_InManual";	//Gr.InManual
// temporare
      AN    #Ma.StStarting;
      ON    #Ma.InManual;
      O     #Ma.CmdOff;	//[4.2]
      R     #Ma.OutStartMan;
      O     #Ma.CmdOn;
      S     #Ma.OutStartMan;
      A     #Ma.CmdNext;
      AN    #Ma.InManual;
      O     #Ma.OutStartMan;
      =     #tmpNext;
      A     #Ma.InManual;
      ON    #Ma.InLocal;
      A(;
      A     #Ma.Par.ParManual;	//[4.1]
      A     #Ma.InManual;
      O     #Ma.InEnable;
      );
      AN    #Ma.CmdOff;
      =     #tmpEnable;
      A     #Ma.InSeqStop;
      AN    #Ma.InManual;
      =     #tmpSeqStop;
//--- Fault----
      A     #RollsLowLeft.StFault;
      O     #RollsUpLeft.StFault;
      O     #RollsLowRight.StFault;
      O     #RollsUpRight.StFault;
      =     #tmpWarning;
      A     #tmpWarning;
      AN    #Ma.Par.ParWarning;
      O     #HLMidLeft.StFault;
      O     #HLInletLeft.StFault;
      O     #SpeedLeft.StFault;
      O     #HLMidRight.StFault;
      O     #HLInletRight.StFault;
      O     #SpeedRight.StFault;
      =     #tmpFaultSum;
//--- Next
      A     #tmpNext;
      S     #RollsLowLeft.CmdNext;
      S     #RollsUpLeft.CmdNext;
      A     #RollsLowLeft.StStartedFwd;
      A     #Ma.Par.Par4Rolls;
      O     #RollsUpLeft.StStartedFwd;
      O     #Ma.InDisableLeft;
      A     #tmpNext;
      S     #RollsLowRight.CmdNext;
      S     #RollsUpRight.CmdNext;
//--- Interlocking Motors
//RollsLowLeft
      A     #tmpEnable;
      AN    #Ma.InDisableLeft;
      =     #RollsLowLeft.InEnableFwd;
// 
      A     #tmpSeqStop;
      =     #RollsLowLeft.InSeqStop;
//RollsUpLeft
      A     #RollsLowLeft.StStartedFwd;
      AN    #Ma.InDisableLeft;
      A     #tmpEnable;
      =     #RollsUpLeft.InEnableFwd;
      A     #tmpSeqStop;
      =     #RollsUpLeft.InSeqStop;
//RollsLowRight
      A     #tmpEnable;
      AN    #Ma.InDisableRight;
      =     #RollsLowRight.InEnableFwd;
// 
      A     #tmpSeqStop;
      =     #RollsLowRight.InSeqStop;
//RollsUpRight
      A     #RollsLowRight.StStartedFwd;
      AN    #Ma.InDisableRight;
      A     #tmpEnable;
      =     #RollsUpRight.InEnableFwd;
      A     #tmpSeqStop;
      =     #RollsUpRight.InSeqStop;
// 
//--- Local mode --
      A     #Ma.InLocal;
      AN    #Ma.InManual;
      =     #RollsLowLeft.InLocal;
      =     #RollsUpLeft.InLocal;
      =     #HLMidLeft.InLocal;
      =     #SpeedLeft.InLocal;
      =     #RollsLowRight.InLocal;
      =     #RollsUpRight.InLocal;
      =     #HLMidRight.InLocal;
      =     #SpeedRight.InLocal;
      =     #HLInletLeft.InLocal;
      =     #HLInletRight.InLocal;
//--- Fault Reset -------------
      A     #Ma.CmdFaultReset;
      S     #RollsLowLeft.CmdFaultReset;
      S     #RollsUpLeft.CmdFaultReset;
      S     #HLMidLeft.CmdFaultReset;
      S     #HLInletLeft.CmdFaultReset;
      S     #SpeedLeft.CmdFaultReset;
      S     #RollsLowRight.CmdFaultReset;
      S     #RollsUpRight.CmdFaultReset;
      S     #HLMidRight.CmdFaultReset;
      S     #HLInletRight.CmdFaultReset;
      S     #SpeedRight.CmdFaultReset;
// 
//--- Monitoring 
      SET;
      S     #HLMidLeft.InMonFalse;
      S     #HLMidRight.InMonFalse;
      AN    #Ma.InOverwriteHL;	//[3.1]
      =     #HLInletLeft.InMonFalse;	//[3.1]
      =     #HLInletRight.InMonFalse;	//[3.1]
      A     #Ma.InpPressureLeft;
      =     #SpeedLeft.InMonTrue;
      A     #Ma.InpPressureRight;
      =     #SpeedRight.InMonTrue;
//Startup done
      A     #RollsLowLeft.StStartedFwd;
      O     #RollsLowLeft.StFault;
      A(;
      A     #RollsUpLeft.StStartedFwd;
      O     #RollsUpLeft.StFault;
      O     #Ma.Par.Par4Rolls;
      );
      O     #Ma.InDisableLeft;
      A(;
      O     #RollsLowRight.StStartedFwd;
      O     #RollsLowRight.StFault;
      O     #Ma.InDisableRight;
      );
      A(;
      O     #RollsUpRight.StStartedFwd;
      O     #RollsUpRight.StFault;
      O     #Ma.InDisableRight;
      O     #Ma.Par.Par4Rolls;
      );
      =     #Ma.OutStartupDone;
      A     #RollsUpLeft.StStartedFwd;
      O     #Ma.Par.Par4Rolls;
      A     #RollsLowLeft.StStartedFwd;
      O     #Ma.InDisableLeft;
      A(;
      A     #RollsUpRight.StStartedFwd;
      O     #Ma.Par.Par4Rolls;	//[3.2]
      A     #RollsLowRight.StStartedFwd;
      O     #Ma.InDisableRight;
      );
      A(;
      ON    #Ma.InDisableLeft;
      ON    #Ma.InDisableRight;
      );
      =     #tmpStarted;
NETWORK
TITLE = Call RollsLowLeft
      CALL  #RollsLowLeft;
NETWORK
TITLE = Call RollsUpLeft
      A     #Ma.Par.Par4Rolls;
      JC    elL3;
      CALL  #RollsUpLeft;
NETWORK
TITLE = Call Digital Input: HLMidLeft
elL3: A     #Ma.Par.Par4Rolls;
      JC    elL4;
      CALL  #HLMidLeft;
NETWORK
TITLE = Call Digital Input: HLInletLeft
elL4: AN    #Ma.Par.ParWithHLInletLeft;
      JC    elL5;
      CALL  #HLInletLeft;
NETWORK
TITLE = Call Digital Input: SMLeft
elL5: AN    #Ma.Par.ParWithSMLeft;
      JC    elL7;
      CALL  #SpeedLeft;
NETWORK
TITLE = Call RollsLowRight
elL7: CALL  #RollsLowRight;
NETWORK
TITLE = Call RollsUpRight
      A     #Ma.Par.Par4Rolls;
      JC    elR3;
      CALL  #RollsUpRight;
NETWORK
TITLE = Call Digital Input: HLMidRight
elR3: A     #Ma.Par.Par4Rolls;
      JC    elR4;
      CALL  #HLMidRight;
NETWORK
TITLE = Call Digital Input: HLInletRight
elR4: AN    #Ma.Par.ParWithHLInletRight;
      JC    elR5;
      CALL  #HLInletRight;
NETWORK
TITLE = Call Digital Input: SMRight
elR5: AN    #Ma.Par.ParWithSMRight;
      JC    StJ0;
      CALL  #SpeedRight;
NETWORK
TITLE = Actual State
// StFault
StJ0: A     #tmpFaultSum;
      =     #Ma.StFault;
// StWarning
      A     #tmpWarning;
      A     #Ma.Par.ParWarning;
      AN    #Ma.StFault;
      =     #Ma.StWarning;
// StStopped
      A     #RollsUpLeft.StStopped;
      O     #Ma.Par.Par4Rolls;
      A(;
      A     #RollsUpRight.StStopped;
      O     #Ma.Par.Par4Rolls;
      );
      A     #RollsLowLeft.StStopped;
      A     #RollsLowRight.StStopped;
      AN    #Ma.StFault;
      =     #Ma.StStopped;
// StStarted
      A     #tmpStarted;
      AN    #Ma.StFault;
      AN    #Ma.StStopped;
      =     #Ma.StStarted;
// StStopping
      A     #RollsLowLeft.InSeqStop;
      O     #RollsLowRight.InSeqStop;
      AN    #Ma.StStarted;
      AN    #Ma.StStopped;
      AN    #Ma.StFault;
      AN    #Ma.StWarning;
      =     #Ma.StStopping;
// StStarting
      AN    #Ma.StStopped;
      AN    #Ma.StStarted;
      AN    #Ma.StStopping;
      AN    #Ma.StFault;
      AN    #Ma.StWarning;
      =     #Ma.StStarting;
NETWORK
TITLE = State Code
// State     StCode
// ----------------------
// StFault32
// StStopped    1
// StStarting   2
// StStarted   3
// StStopping  7
// StWarning8
      A     #Ma.StStopped;
      L     1;	//Code=StStopped
      JC    Code;
      A     #Ma.StStarted;
      L     3;	//Code=StStarted
      JC    Code;
      A     #Ma.StWarning;
      L     8;	//Code=StWarning 
      JC    Code;
      A     #Ma.StStarting;
      L     2;	//Code=StStarting
      JC    Code;
      A     #Ma.StStopping;
      L     7;	//Code=StStopping 
      JC    Code;
      L     32;	//Code=StFault 
Code: L     #Ma.StCode;	// Old state code
      TAK;
      T     #Ma.StCode;	// Save state code
      <>I;
      L     3;
      CC    "SYS_CBitCtrl";	//Set change bit
NETWORK
TITLE = Global End
      CLR;	//---Clear all commands
      =     #Ma.CmdOn;
      =     #Ma.CmdOff;
      =     #Ma.CmdNext;
      =     #Ma.CmdFaultReset;
END_FUNCTION_BLOCK

FUNCTION_BLOCK "GCS7_M_PelletCooler"	// FB 47
TITLE = Pellet Cooler
//  
//COPYRIGHT:    (C) 1997  BUHLER AG, CH-9240 UZWIL,  SWITZERLAND
//
//PRODUCT:      GCS7
//
//TITLE:        FB 47 Machine Control:Pellet Coller 
//
//-------------------------------------------------------------------------
//
//IDENT:        AUTHOR:             DEPT:                       DATE:
//
//FB47.4.0      A. Egli             CT3                         17-Jun-2002
//              New Release with one block 
//FB47.3.0      A. Egli             CT3                         11-Oct-1999
//              Local data reduced 
//FB47.2C       K. Tischer          MU664                       06-Mrz-1999
//              Transition to StEmptying only if tmpEnable
//FB47.2B       K. Tischer          MU664                       06-Mrz-1999
//              CC FC2 not UC FC2
//FB47.2A       A. Egli             CT3                         04-Mai-1998
//              StFault = StCode 32
//FB47.1A       A.Egli              AEE61                       12-Nov-1997
//              1st Release in S7
//
//-------------------------------------------------------------------------
//
//PURPOSE:      MANUAL : see [LL.PTCxxMAN]
//
//RESTRICTIONS: S7
//              ACCU2: Pointer to dynamic datas of the machine
//              ACCU1: Pointer to parameter datas of the machine
//
//-------------------------------------------------------------------------
//
//
AUTHOR : EA
FAMILY : GCS7LL
NAME : PelletCo
VERSION : 4.0
VAR
  Ma : UDT 20470;
  Slide : FB 20;	//Element
  Motor : FB 12;	//Element
  Level : FB 14;	//Element
END_VAR
VAR_TEMP
  tmpFaultStop : BOOL ;
  tmpFaultSum : BOOL ;
  tmpNext : BOOL ;
  tmpLocal : BOOL ;
  tmpEnable : BOOL ;
  tmpEnableOpen : BOOL ;
  tmpEmpty : BOOL ;
  tmpLenDyn : INT ;
END_VAR
BEGIN
NETWORK
TITLE =
      L     16;
      T     #tmpLenDyn;
NETWORK
TITLE = PC Control
//=== Test Object number =====================
      L     "SYS_DirectCtrlDB".PC.ObjectNo;	//"SYS_PCControl".ObjectNo
      L     #Ma.Par.ParObjectNo;	//Input ObjectNo
      <>I;
      JC    aEnd;
//=== Test OType      ========================
      L     2047;	//Input object type
      L     "SYS_DirectCtrlDB".PC.ObjectType;	//"SYS_PCControl".ObjectType
      <>I;
      JC    aEnd;
//=== Test Handshake =========================
      A     "SYS_DirectCtrlDB".PC.Hsk.FExamine;	// Handshake.FExamine
      JC    aExa;
      A     "SYS_DirectCtrlDB".PC.Hsk.FDefineCmd;	// Handshake.FDefineCmd
      JC    aCmd;
      A     "SYS_DirectCtrlDB".PC.Hsk.FDefinePara;	// Handshake.FDefinePara
      JC    pPar;
aIni: L     2;	// FcInit
      UC    "SYS_DirectCtrl";
      JU    aEnd;
// Write parameter 
pPar: LAR1  P#DBX 58.0;
      L     P#6.0;
      +AR1;
      L     DBW [AR1,P#4.0];
      T     #Ma.Par.ParEmptyingTime;
// Write new commands from PC to Interface of group 
aCmd: A     "SYS_DirectCtrlDB".PC.Cmd1[8];	//Cmd1[8]=CmdOff
      S     #Ma.CmdOff;
      A     "SYS_DirectCtrlDB".PC.Cmd1[9];	//Cmd1[9]=CmdOn
      S     #Ma.CmdOn;
      A     "SYS_DirectCtrlDB".PC.Cmd1[10];	//Cmd1[10]=CmdNext
      S     #Ma.CmdNext;
      A     "SYS_DirectCtrlDB".PC.Cmd1[11];	//Cmd1[11]=CmdFaultReset
      S     #Ma.CmdFaultReset;
      A     "SYS_DirectCtrlDB".PC.Cmd1[13];	//Cmd1[13]=CmdManualOn
      S     #Ma.InManual;
      A     "SYS_DirectCtrlDB".PC.Cmd2[13];	//Cmd1[13]=CmdManualOff
      R     #Ma.InManual;
      A     "SYS_DirectCtrlDB".PC.Cmd1[1];	//Cmd1[1]=CmdMiddle1
      S     #Ma.InMiddle1;
      R     #Ma.InMiddle2;
      R     #Ma.InFullOpen;
      R     #Ma.InEmptying;
      S     #Ma.CmdOn;
      A     "SYS_DirectCtrlDB".PC.Cmd1[2];	//Cmd1[2]=CmdMiddle2
      R     #Ma.InMiddle1;
      S     #Ma.InMiddle2;
      R     #Ma.InFullOpen;
      R     #Ma.InEmptying;
      S     #Ma.CmdOn;
      A     "SYS_DirectCtrlDB".PC.Cmd1[3];	//Cmd1[3]=CmdFullOpen
      R     #Ma.InMiddle1;
      R     #Ma.InMiddle2;
      S     #Ma.InFullOpen;
      R     #Ma.InEmptying;
      S     #Ma.CmdOn;
      A     "SYS_DirectCtrlDB".PC.Cmd1[4];	//Cmd1[4]=CmdEmptying
      S     #Ma.InEmptying;
      S     #Ma.CmdOn;
      A     "SYS_DirectCtrlDB".PC.Cmd1[5];	//Cmd1[5]=CmdRestDischarge
      S     #Ma.CmdRestdischarge;
      JU    aIni;
aExa: TAR2;	// Address Dynamic data
      T     "SYS_DirectCtrlDB".GC.InDynAddr;	// -->"SYS_PCControl".GC.InDynAddr
      L     #tmpLenDyn;	// Length Dynamic data
      T     "SYS_DirectCtrlDB".GC.InDynLen;	// -->PCControl.GC.InDynLen
      L     0;
      T     "SYS_DirectCtrlDB".GC.InParaAddr;	// -->PCControl.GC.InParaAddr
      T     "SYS_DirectCtrlDB".GC.InParaLen;	// -->PCControl.GC.InParaLen
      L     1;	// Code FcExamine
      UC    "SYS_DirectCtrl";
      L     10;	//Revision
      T     "SYS_DirectCtrlDB".GC.Revision;
aEnd: NOP   0;
NETWORK
TITLE = Interlocking
//===Global Group Orders===
      A     "GCS7_Gr_OutManualOn";	//Gr.OutManualOn
      S     #Ma.InManual;
      A     "GCS7_Gr_OutManualOff";	//Gr.OutManualOff
      R     #Ma.InManual;
      A     #Ma.InManual;
      S     "GCS7_Gr_InManual";	//Gr.InManual
      A     #Ma.CmdNext;
      AN    #Ma.InManual;
      O     #Ma.CmdOn;
      =     #tmpNext;
      A     #Ma.InManual;
      ON    #Ma.InLocal;
      A     #Ma.InEnable;
      AN    #Ma.CmdOff;
      =     #tmpEnable;
//--- Fault----
      A     #Slide.StFault;
      O     #Level.StFault;
      O     #Motor.StFault;
      =     #tmpFaultSum;
//--- Next
      A     #Ma.InManual;
      AN    #Slide.StLN;
      O     #tmpNext;
      S     #Motor.CmdNext;
//--- Interlocking Motor
      AN    #Slide.StLN;
      AN    #Slide.StFault;
      A     #tmpEnable;
      =     #Motor.InEnableFwd;
//--- Interlocking Slide
//    Close
      A     #Level.StFalse;
      A     #Ma.Par.ParWithLevel;
      AN    #Ma.InManual;
      AN    #Ma.InEmptying;
      AN    #Ma.StEmptying;
      O     #Ma.StEmptied;
      ON    #tmpEnable;
      O     #Ma.StStopping;
      =     #Slide.InLN;
//    Opening
      AN    #Ma.Par.ParWithLevel;
      O     #Level.StTrue;	//Covered
      O     #Ma.InManual;
      O     #Ma.StEmptying;
      A     #tmpNext;
      AN    #Slide.InLN;
      =     #tmpEnableOpen;
//    Full Open
      A     #Ma.Par.ParAutoRestDischarge;
      O     #Ma.CmdRestdischarge;
      S     #Ma.OutRestDischarge;
      AN    #Ma.StEmptying;
      ON    #Ma.OutEmptyingTimeDone;
      R     #Ma.OutRestDischarge;
      A     #Ma.OutRestDischarge;
      O     #Ma.InFullOpen;
      A     #tmpEnableOpen;
      S     #Slide.CmdHN;
//    Middle 1
      A     #tmpEnableOpen;
      AN    #Slide.CmdHN;
      A     #Ma.InMiddle1;
      S     #Slide.CmdMiddle1;
//    Middle 2
      A     #tmpEnableOpen;
      AN    #Slide.CmdHN;
      A     #Ma.InMiddle2;
      S     #Slide.CmdMiddle2;
// 
//--- Local mode --
      A     #Ma.InLocal;
      AN    #Ma.InManual;
      =     #Slide.InLocal;
      =     #Level.InLocal;
      =     #Motor.InLocal;
//--- Fault Reset -------------
      A     #Ma.CmdFaultReset;
      S     #Slide.CmdFaultReset;
      S     #Level.CmdFaultReset;
      S     #Motor.CmdFaultReset;
// 
//--- Monitoring Level
NETWORK
TITLE = Call Slide
      CALL  #Slide;
NETWORK
TITLE = Call Digital Input: Level
      AN    #Ma.Par.ParWithLevel;
      JC    el4;
      CALL  #Level;
NETWORK
TITLE = Call Motor
el4:  CALL  #Motor;
NETWORK
TITLE = Jump to actual state
      A     #Ma.StStopped;
      JC    S0;	// ===> State
      A     #Ma.StStarted;
      JC    S2;	// ===> State
      A     #Ma.StStarting;
      JC    S1;	// ===> State
      A     #Ma.StStopping;
      JC    S3;	// ===> State
      A     #Ma.StFault;
      JC    S4;	// ===> State
      A     #Ma.StEmptying;
      JC    S5;	// ===> State
      A     #Ma.StEmptied;
      JC    S6;	// ===> State
NETWORK
TITLE = Stopped
//any Transition 
xxS0: S     #Ma.StStopped;	// ===> Initialisation
//=== Logic
// Condition for StFault
S0:   A     #tmpFaultSum;
      R     #Ma.StStopped;
      JC    xxS4;	//--> ST_FAULT:
// Condition for StStarting
      A     #tmpNext;
      A     #tmpEnable;
      ON    #Motor.StStopped;
      ON    #Slide.StLN;
      R     #Ma.StStopped;
      JC    xxS1;	//--> StStarting
      JU    OUT;
NETWORK
TITLE = StStarting
//any Transition 
xxS1: S     #Ma.StStarting;
//=== Logic
// Condition for StFault
S1:   A     #tmpFaultSum;
      R     #Ma.StStarting;
      JC    xxS4;	//--> StFault
// Condition for StEmptying
      A     #Ma.InEmptying;
      A     #tmpEnable;	//[Rel 2C]
      R     #Ma.StStarting;
      JC    xxS5;	//--> StEmptying
// Condition for StStarted
      A     #Motor.StStartedFwd;
      AN    #Slide.StLN;
      O;
      A     #Ma.Par.ParWithLevel;
      AN    #Level.StTrue;	//Covered
      R     #Ma.StStarting;
      JC    xxS2;	//-->StStarted
// Condition for StStopping
      AN    #tmpEnable;
      AN    #Motor.StStartedFwd;
      R     #Ma.StStarting;
      JC    xxS3;	//-->StStopping
      JU    OUT;
NETWORK
TITLE = StStarted
//any Transition 
xxS2: S     #Ma.StStarted;
//=== Logic
// Condition for StFault
S2:   A     #tmpFaultSum;
      R     #Ma.StStarted;
      JC    xxS4;	//--> StFault
// Condition for StEmptying
      A     #Ma.InEmptying;
      A     #tmpEnable;	//[Rel 2C]
      R     #Ma.StStarted;
      JC    xxS5;	//--> StEmptying
// Condition for StStopping
      AN    #tmpEnable;
      AN    #Motor.StStartedFwd;
      R     #Ma.StStarted;
      JC    xxS3;	//-->StStopping
      JU    OUT;
NETWORK
TITLE = Stopping
//any Transition 
xxS3: S     #Ma.StStopping;
//=== Logic
// Condition for StFault
S3:   A     #tmpFaultSum;
      R     #Ma.StStopping;
      JC    xxS4;	//--> StFault
// Condition for StStopped
      A     #Motor.StStopped;
      A     #Slide.StLN;
      R     #Ma.StStopping;
      JC    xxS0;	//-->StStopped
// Condition for StStarting
      A     #Motor.StStartedFwd;
      AN    #Slide.StLN;
      R     #Ma.StStopping;
      JC    xxS1;	//-->StStarting
      JU    OUT;
NETWORK
TITLE = Fault
//any Transition 
xxS4: S     #Ma.StFault;
      JU    OUT;
//=== Logic
S4:   A     #tmpFaultSum;
      JC    OUT;
//---- Transition --
      R     #Ma.StFault;
      JU    xxS0;	//-->StStopping 
NETWORK
TITLE = StEmptying
//any Transition 
xxS5: S     #Ma.StEmptying;
      L     #Ma.Par.ParEmptyingTime;
      T     #Ma.Par.OutEmptyingTime;
//=== Logic
// Condition for StFault
S5:   A     #tmpFaultSum;
      R     #Ma.StEmptying;
      R     #Ma.OutEmptyingTimeDone;
      JC    xxS4;	//--> StFault
// Condition for StEmptied
      L     #Ma.Par.OutEmptyingTime;
      ON    #Motor.StStartedFwd;
      ON    "GCS7_Gr_OutTick500ms";	//Gr.OutTick500ms
      O;
      A     #Level.StTrue;
      A     #Ma.Par.ParWithLevel;
      O     #Ma.OutEmptyingTimeDone;
      JC    S5J1;
      +     -5;
      T     #Ma.Par.OutEmptyingTime;
S5J1: L     0;
      <=I;
      =     #Ma.OutEmptyingTimeDone;
      A     #Slide.StHN;
      AN    #Slide.Par.OutPulseIsOn;
      A     #Ma.OutEmptyingTimeDone;
      R     #Ma.OutEmptyingTimeDone;
      R     #Ma.StEmptying;
      JC    xxS6;	//-->StEmptied
// Condition for StStopping
      AN    #Ma.InEmptying;
      ON    #tmpEnable;
      R     #Ma.OutEmptyingTimeDone;
      R     #Ma.StEmptying;
      JC    xxS3;	//-->StStopping
      JU    OUT;
NETWORK
TITLE = StEmptied
//any Transition 
xxS6: S     #Ma.StEmptied;
      JU    OUT;
//=== Logic
// Condition for StFault
S6:   A     #tmpFaultSum;
      R     #Ma.StEmptied;
      JC    xxS4;	//--> StFault
// Condition for StStopping
      AN    #Ma.InEmptying;
      R     #Ma.StEmptied;
      JC    xxS1;	//-->StStopping
      JU    OUT;
NETWORK
TITLE = State Code
// State     StCode
// ----------------------
// StFault32
// StStopped    1
// StStarting   2
// StStarted.Wait   3
// StStarted.Feeding4
// StEmptying    5
// StEmptied    6
// StStopping  7
OUT:  A     #Ma.StStopped;
      L     1;	//Code=StStopped
      JC    Code;
      A     #Ma.StStarted;
      A     #Slide.StLN;
      L     3;	//Code=StWaiting
      JC    Code;
      A     #Ma.StStarted;
      L     4;	//Code=StFeeding
      JC    Code;
      A     #Ma.StEmptying;
      L     5;	//Code=StEmptying
      JC    Code;
      A     #Ma.StEmptied;
      L     6;	//Code=StEmptied
      JC    Code;
      A     #Ma.StStarting;
      L     2;	//Code=StStarting
      JC    Code;
      A     #Ma.StStopping;
      L     7;	//Code=StStopping 
      JC    Code;
      L     32;	//Code=StFault 
Code: L     #Ma.StCode;	// Old state code
      TAK;
      T     #Ma.StCode;	// Save state code
      <>I;
      L     3;
      CC    "SYS_CBitCtrl";	//Set change bit
NETWORK
TITLE = Global End
      CLR;	//---Clear all commands
      =     #Ma.CmdOn;
      =     #Ma.CmdOff;
      =     #Ma.CmdNext;
      =     #Ma.CmdFaultReset;
      =     #Ma.CmdRestdischarge;
END_FUNCTION_BLOCK

